Staubli VAL3: Compensated.dtx

public frame fReference = {x=1504.182, y=53.840, z=-415.791, rx=0.201, ry=-0.641, rz=0.004, fatherId=world[0]}
public jointRx jPark = {j1=0.000, j2=0.000, j3=90.000, j4=0.000, j5=90.000, j6=0.000}
public jointRx jJoint = {j1=2.01098, j2=34.80611, j3=88.39690, j4=0.21482, j5=56.14953, j6=-178.11080}
public mdesc mNomSpeed = {accel=100, vel=100, decel=100, tmax=99999, rmax=99999, blend=off, leave=50, reach=50}
public mdesc mSpeed = {tmax=33.3, rmax=100, leave=0.1, reach=0.1, blend=cartesian}
public num nTraj
num nTimeStop
num nTimeStart
num nMode
num nEtat
public pointRx pPoint[1313]
  [0] = {x=-35.000, y=0.000, z=0.000, rx=-0.000, ry=0.000, rz=-0.000, shoulder=lefty, elbow=epositive, wrist=wpositive, fatherId=fReference[0]}
  [1] = {x=-34.500, y=0.000, z=-0.007, rx=-0.000, ry=0.000, rz=-0.000, shoulder=lefty, elbow=epositive, wrist=wpositive, fatherId=fReference[0]}
  [2] = {x=-34.000, y=0.000, z=-0.014, rx=-0.000, ry=0.000, rz=-0.000, shoulder=lefty, elbow=epositive, wrist=wpositive, fatherId=fReference[0]}
  [3] = {x=-33.499, y=0.000, z=-0.022, rx=-0.000, ry=0.000, rz=-0.000, shoulder=lefty, elbow=epositive, wrist=wpositive, fatherId=fReference[0]}
  [4] = {x=-32.998, y=0.000, z=-0.029, rx=-0.000, ry=0.000, rz=-0.000, shoulder=lefty, elbow=epositive, wrist=wpositive, fatherId=fReference[0]}
  [5] = {x=-32.497, y=0.000, z=-0.036, rx=-0.000, ry=0.000, rz=-0.000, shoulder=lefty, elbow=epositive, wrist=wpositive, fatherId=fReference[0]}
  [6] = {x=-31.997, y=0.000, z=-0.044, rx=-0.000, ry=0.000, rz=-0.000, shoulder=lefty, elbow=epositive, wrist=wpositive, fatherId=fReference[0]}
  [7] = {x=-31.496, y=0.000, z=-0.051, rx=-0.000, ry=0.000, rz=-0.000, shoulder=lefty, elbow=epositive, wrist=wpositive, fatherId=fReference[0]}
  [8] = {x=-30.995, y=0.000, z=-0.059, rx=-0.000, ry=0.000, rz=-0.000, shoulder=lefty, elbow=epositive, wrist=wpositive, fatherId=fReference[0]}
  [9] = {x=-30.494, y=0.000, z=-0.066, rx=-0.000, ry=0.000, rz=-0.000, shoulder=lefty, elbow=epositive, wrist=wpositive, fatherId=fReference[0]}
  [10] = {x=-29.993, y=0.000, z=-0.073, rx=-0.000, ry=0.000, rz=-0.000, shoulder=lefty, elbow=epositive, wrist=wpositive, fatherId=fReference[0]}
  [11] = {x=-29.493, y=0.000, z=-0.081, rx=-0.000, ry=0.000, rz=-0.000, shoulder=lefty, elbow=epositive, wrist=wpositive, fatherId=fReference[0]}
  [12] = {x=-28.992, y=0.000, z=-0.088, rx=-0.000, ry=0.000, rz=-0.000, shoulder=lefty, elbow=epositive, wrist=wpositive, fatherId=fReference[0]}
  [13] = {x=-28.491, y=0.000, z=-0.095, rx=-0.000, ry=0.000, rz=-0.000, shoulder=lefty, elbow=epositive, wrist=wpositive, fatherId=fReference[0]}
  [14] = {x=-27.991, y=0.000, z=-0.103, rx=-0.000, ry=0.000, rz=-0.000, shoulder=lefty, elbow=epositive, wrist=wpositive, fatherId=fReference[0]}
  [15] = {x=-27.490, y=0.000, z=-0.110, rx=-0.000, ry=0.000, rz=-0.000, shoulder=lefty, elbow=epositive, wrist=wpositive, fatherId=fReference[0]}
  [16] = {x=-26.989, y=0.000, z=-0.117, rx=-0.000, ry=0.000, rz=-0.000, shoulder=lefty, elbow=epositive, wrist=wpositive, fatherId=fReference[0]}
  [17] = {x=-26.489, y=0.000, z=-0.125, rx=-0.000, ry=0.000, rz=-0.000, shoulder=lefty, elbow=epositive, wrist=wpositive, fatherId=fReference[0]}
  [18] = {x=-25.988, y=0.000, z=-0.132, rx=-0.000, ry=0.000, rz=-0.000, shoulder=lefty, elbow=epositive, wrist=wpositive, fatherId=fReference[0]}
  [19] = {x=-25.487, y=0.000, z=-0.139, rx=-0.000, ry=0.000, rz=-0.000, shoulder=lefty, elbow=epositive, wrist=wpositive, fatherId=fReference[0]}
  [20] = {x=-24.987, y=0.000, z=-0.147, rx=-0.000, ry=0.000, rz=-0.000, shoulder=lefty, elbow=epositive, wrist=wpositive, fatherId=fReference[0]}
  [21] = {x=-24.486, y=0.000, z=-0.154, rx=-0.000, ry=0.000, rz=-0.000, shoulder=lefty, elbow=epositive, wrist=wpositive, fatherId=fReference[0]}
  [22] = {x=-23.986, y=0.000, z=-0.161, rx=-0.000, ry=0.000, rz=-0.000, shoulder=lefty, elbow=epositive, wrist=wpositive, fatherId=fReference[0]}
  [23] = {x=-23.485, y=0.000, z=-0.169, rx=-0.000, ry=0.000, rz=-0.000, shoulder=lefty, elbow=epositive, wrist=wpositive, fatherId=fReference[0]}
  [24] = {x=-22.985, y=0.000, z=-0.176, rx=-0.000, ry=0.000, rz=-0.000, shoulder=lefty, elbow=epositive, wrist=wpositive, fatherId=fReference[0]}
  [25] = {x=-22.484, y=0.000, z=-0.183, rx=-0.000, ry=0.000, rz=-0.000, shoulder=lefty, elbow=epositive, wrist=wpositive, fatherId=fReference[0]}
  [26] = {x=-21.983, y=0.000, z=-0.191, rx=-0.000, ry=0.000, rz=-0.000, shoulder=lefty, elbow=epositive, wrist=wpositive, fatherId=fReference[0]}
  [27] = {x=-21.483, y=0.000, z=-0.198, rx=-0.000, ry=0.000, rz=-0.000, shoulder=lefty, elbow=epositive, wrist=wpositive, fatherId=fReference[0]}
  [28] = {x=-20.982, y=0.000, z=-0.205, rx=-0.000, ry=0.000, rz=-0.000, shoulder=lefty, elbow=epositive, wrist=wpositive, fatherId=fReference[0]}
  [29] = {x=-20.482, y=0.000, z=-0.213, rx=-0.000, ry=0.000, rz=-0.000, shoulder=lefty, elbow=epositive, wrist=wpositive, fatherId=fReference[0]}
  [30] = {x=-19.981, y=0.000, z=-0.220, rx=-0.000, ry=0.000, rz=-0.000, shoulder=lefty, elbow=epositive, wrist=wpositive, fatherId=fReference[0]}
  [31] = {x=-19.481, y=0.000, z=-0.227, rx=-0.000, ry=0.000, rz=-0.000, shoulder=lefty, elbow=epositive, wrist=wpositive, fatherId=fReference[0]}
  [32] = {x=-18.980, y=0.000, z=-0.234, rx=-0.000, ry=0.000, rz=-0.000, shoulder=lefty, elbow=epositive, wrist=wpositive, fatherId=fReference[0]}
  [33] = {x=-18.480, y=0.000, z=-0.242, rx=-0.000, ry=0.000, rz=-0.000, shoulder=lefty, elbow=epositive, wrist=wpositive, fatherId=fReference[0]}
  [34] = {x=-17.979, y=0.000, z=-0.249, rx=-0.000, ry=0.000, rz=-0.000, shoulder=lefty, elbow=epositive, wrist=wpositive, fatherId=fReference[0]}
  [35] = {x=-17.479, y=0.000, z=-0.256, rx=-0.000, ry=0.000, rz=-0.000, shoulder=lefty, elbow=epositive, wrist=wpositive, fatherId=fReference[0]}
  [36] = {x=-16.978, y=0.000, z=-0.264, rx=-0.000, ry=0.000, rz=-0.000, shoulder=lefty, elbow=epositive, wrist=wpositive, fatherId=fReference[0]}
  [37] = {x=-16.478, y=0.000, z=-0.271, rx=-0.000, ry=0.000, rz=-0.000, shoulder=lefty, elbow=epositive, wrist=wpositive, fatherId=fReference[0]}
  [38] = {x=-15.977, y=0.000, z=-0.278, rx=-0.000, ry=0.000, rz=-0.000, shoulder=lefty, elbow=epositive, wrist=wpositive, fatherId=fReference[0]}
  [39] = {x=-15.477, y=0.000, z=-0.285, rx=-0.000, ry=0.000, rz=-0.000, shoulder=lefty, elbow=epositive, wrist=wpositive, fatherId=fReference[0]}
  [40] = {x=-14.976, y=0.000, z=-0.293, rx=-0.000, ry=0.000, rz=-0.000, shoulder=lefty, elbow=epositive, wrist=wpositive, fatherId=fReference[0]}
  [41] = {x=-14.476, y=0.000, z=-0.300, rx=-0.000, ry=0.000, rz=-0.000, shoulder=lefty, elbow=epositive, wrist=wpositive, fatherId=fReference[0]}
  [42] = {x=-13.975, y=0.000, z=-0.307, rx=-0.000, ry=0.000, rz=-0.000, shoulder=lefty, elbow=epositive, wrist=wpositive, fatherId=fReference[0]}
  [43] = {x=-13.475, y=0.000, z=-0.315, rx=-0.000, ry=0.000, rz=-0.000, shoulder=lefty, elbow=epositive, wrist=wpositive, fatherId=fReference[0]}
  [44] = {x=-12.975, y=0.000, z=-0.322, rx=-0.000, ry=0.000, rz=-0.000, shoulder=lefty, elbow=epositive, wrist=wpositive, fatherId=fReference[0]}
  [45] = {x=-12.474, y=0.000, z=-0.329, rx=-0.000, ry=0.000, rz=-0.000, shoulder=lefty, elbow=epositive, wrist=wpositive, fatherId=fReference[0]}
  [46] = {x=-11.974, y=0.000, z=-0.336, rx=-0.000, ry=0.000, rz=-0.000, shoulder=lefty, elbow=epositive, wrist=wpositive, fatherId=fReference[0]}
  [47] = {x=-11.473, y=0.000, z=-0.344, rx=-0.000, ry=0.000, rz=-0.000, shoulder=lefty, elbow=epositive, wrist=wpositive, fatherId=fReference[0]}
  [48] = {x=-10.973, y=0.000, z=-0.351, rx=-0.000, ry=0.000, rz=-0.000, shoulder=lefty, elbow=epositive, wrist=wpositive, fatherId=fReference[0]}
  [49] = {x=-10.472, y=0.000, z=-0.358, rx=-0.000, ry=0.000, rz=-0.000, shoulder=lefty, elbow=epositive, wrist=wpositive, fatherId=fReference[0]}
  [50] = {x=-9.972, y=0.000, z=-0.366, rx=-0.000, ry=0.000, rz=-0.000, shoulder=lefty, elbow=epositive, wrist=wpositive, fatherId=fReference[0]}
  [51] = {x=-9.471, y=0.000, z=-0.373, rx=-0.000, ry=0.000, rz=-0.000, shoulder=lefty, elbow=epositive, wrist=wpositive, fatherId=fReference[0]}
  [52] = {x=-8.971, y=0.000, z=-0.380, rx=-0.000, ry=0.000, rz=-0.000, shoulder=lefty, elbow=epositive, wrist=wpositive, fatherId=fReference[0]}
  [53] = {x=-8.470, y=0.000, z=-0.388, rx=-0.000, ry=0.000, rz=-0.000, shoulder=lefty, elbow=epositive, wrist=wpositive, fatherId=fReference[0]}
  [54] = {x=-7.969, y=0.000, z=-0.395, rx=-0.000, ry=0.000, rz=-0.000, shoulder=lefty, elbow=epositive, wrist=wpositive, fatherId=fReference[0]}
  [55] = {x=-7.469, y=0.000, z=-0.402, rx=-0.000, ry=0.000, rz=-0.000, shoulder=lefty, elbow=epositive, wrist=wpositive, fatherId=fReference[0]}
  [56] = {x=-6.968, y=0.000, z=-0.409, rx=-0.000, ry=0.000, rz=-0.000, shoulder=lefty, elbow=epositive, wrist=wpositive, fatherId=fReference[0]}
  [57] = {x=-6.468, y=0.000, z=-0.417, rx=-0.000, ry=0.000, rz=-0.000, shoulder=lefty, elbow=epositive, wrist=wpositive, fatherId=fReference[0]}
  [58] = {x=-5.967, y=0.000, z=-0.424, rx=-0.000, ry=0.000, rz=-0.000, shoulder=lefty, elbow=epositive, wrist=wpositive, fatherId=fReference[0]}
  [59] = {x=-5.467, y=0.000, z=-0.431, rx=-0.000, ry=0.000, rz=-0.000, shoulder=lefty, elbow=epositive, wrist=wpositive, fatherId=fReference[0]}
  [60] = {x=-4.966, y=0.000, z=-0.439, rx=-0.000, ry=0.000, rz=-0.000, shoulder=lefty, elbow=epositive, wrist=wpositive, fatherId=fReference[0]}
  [61] = {x=-4.466, y=0.000, z=-0.446, rx=-0.000, ry=0.000, rz=-0.000, shoulder=lefty, elbow=epositive, wrist=wpositive, fatherId=fReference[0]}
  [62] = {x=-3.965, y=0.000, z=-0.453, rx=-0.000, ry=0.000, rz=-0.000, shoulder=lefty, elbow=epositive, wrist=wpositive, fatherId=fReference[0]}
  [63] = {x=-3.464, y=0.000, z=-0.461, rx=-0.000, ry=0.000, rz=-0.000, shoulder=lefty, elbow=epositive, wrist=wpositive, fatherId=fReference[0]}
  [64] = {x=-2.964, y=0.000, z=-0.468, rx=-0.000, ry=0.000, rz=-0.000, shoulder=lefty, elbow=epositive, wrist=wpositive, fatherId=fReference[0]}
  [65] = {x=-2.463, y=0.000, z=-0.475, rx=-0.000, ry=0.000, rz=-0.000, shoulder=lefty, elbow=epositive, wrist=wpositive, fatherId=fReference[0]}
  [66] = {x=-1.963, y=0.000, z=-0.483, rx=-0.000, ry=0.000, rz=-0.000, shoulder=lefty, elbow=epositive, wrist=wpositive, fatherId=fReference[0]}
  [67] = {x=-1.462, y=0.000, z=-0.490, rx=-0.000, ry=0.000, rz=-0.000, shoulder=lefty, elbow=epositive, wrist=wpositive, fatherId=fReference[0]}
  [68] = {x=-0.961, y=0.000, z=-0.497, rx=-0.000, ry=0.000, rz=-0.000, shoulder=lefty, elbow=epositive, wrist=wpositive, fatherId=fReference[0]}
  [69] = {x=-0.461, y=0.000, z=-0.505, rx=-0.000, ry=0.000, rz=-0.000, shoulder=lefty, elbow=epositive, wrist=wpositive, fatherId=fReference[0]}
  [70] = {x=0.040, y=0.000, z=-0.512, rx=-0.000, ry=0.000, rz=-0.000, shoulder=lefty, elbow=epositive, wrist=wpositive, fatherId=fReference[0]}
  [71] = {x=0.541, y=0.000, z=-0.519, rx=-0.000, ry=0.000, rz=-0.000, shoulder=lefty, elbow=epositive, wrist=wpositive, fatherId=fReference[0]}
  [72] = {x=1.041, y=0.000, z=-0.527, rx=-0.000, ry=0.000, rz=-0.000, shoulder=lefty, elbow=epositive, wrist=wpositive, fatherId=fReference[0]}
  [73] = {x=1.542, y=0.000, z=-0.534, rx=-0.000, ry=0.000, rz=-0.000, shoulder=lefty, elbow=epositive, wrist=wpositive, fatherId=fReference[0]}
  [74] = {x=2.043, y=0.000, z=-0.541, rx=-0.000, ry=0.000, rz=-0.000, shoulder=lefty, elbow=epositive, wrist=wpositive, fatherId=fReference[0]}
  [75] = {x=2.544, y=0.000, z=-0.549, rx=-0.000, ry=0.000, rz=-0.000, shoulder=lefty, elbow=epositive, wrist=wpositive, fatherId=fReference[0]}
  [76] = {x=3.044, y=0.000, z=-0.556, rx=-0.000, ry=0.000, rz=-0.000, shoulder=lefty, elbow=epositive, wrist=wpositive, fatherId=fReference[0]}
  [77] = {x=3.545, y=0.000, z=-0.563, rx=-0.000, ry=0.000, rz=-0.000, shoulder=lefty, elbow=epositive, wrist=wpositive, fatherId=fReference[0]}
  [78] = {x=4.046, y=0.000, z=-0.571, rx=-0.000, ry=0.000, rz=-0.000, shoulder=lefty, elbow=epositive, wrist=wpositive, fatherId=fReference[0]}
  [79] = {x=4.547, y=0.000, z=-0.578, rx=-0.000, ry=0.000, rz=-0.000, shoulder=lefty, elbow=epositive, wrist=wpositive, fatherId=fReference[0]}
  [80] = {x=5.047, y=0.000, z=-0.586, rx=-0.000, ry=0.000, rz=-0.000, shoulder=lefty, elbow=epositive, wrist=wpositive, fatherId=fReference[0]}
  [81] = {x=5.548, y=0.000, z=-0.593, rx=-0.000, ry=0.000, rz=-0.000, shoulder=lefty, elbow=epositive, wrist=wpositive, fatherId=fReference[0]}
  [82] = {x=6.049, y=0.000, z=-0.600, rx=-0.000, ry=0.000, rz=-0.000, shoulder=lefty, elbow=epositive, wrist=wpositive, fatherId=fReference[0]}
  [83] = {x=6.550, y=0.000, z=-0.608, rx=-0.000, ry=0.000, rz=-0.000, shoulder=lefty, elbow=epositive, wrist=wpositive, fatherId=fReference[0]}
  [84] = {x=7.051, y=0.000, z=-0.615, rx=-0.000, ry=0.000, rz=-0.000, shoulder=lefty, elbow=epositive, wrist=wpositive, fatherId=fReference[0]}
  [85] = {x=7.552, y=0.000, z=-0.623, rx=-0.000, ry=0.000, rz=-0.000, shoulder=lefty, elbow=epositive, wrist=wpositive, fatherId=fReference[0]}
  [86] = {x=8.053, y=0.000, z=-0.630, rx=-0.000, ry=0.000, rz=-0.000, shoulder=lefty, elbow=epositive, wrist=wpositive, fatherId=fReference[0]}
  [87] = {x=8.554, y=0.000, z=-0.637, rx=-0.000, ry=0.000, rz=-0.000, shoulder=lefty, elbow=epositive, wrist=wpositive, fatherId=fReference[0]}
  [88] = {x=9.055, y=0.000, z=-0.645, rx=-0.000, ry=0.000, rz=-0.000, shoulder=lefty, elbow=epositive, wrist=wpositive, fatherId=fReference[0]}
  [89] = {x=9.556, y=0.000, z=-0.652, rx=-0.000, ry=0.000, rz=-0.000, shoulder=lefty, elbow=epositive, wrist=wpositive, fatherId=fReference[0]}
  [90] = {x=10.057, y=0.000, z=-0.660, rx=-0.000, ry=0.000, rz=-0.000, shoulder=lefty, elbow=epositive, wrist=wpositive, fatherId=fReference[0]}
  [91] = {x=10.558, y=0.000, z=-0.667, rx=-0.000, ry=0.000, rz=-0.000, shoulder=lefty, elbow=epositive, wrist=wpositive, fatherId=fReference[0]}
  [92] = {x=11.059, y=0.000, z=-0.675, rx=-0.000, ry=0.000, rz=-0.000, shoulder=lefty, elbow=epositive, wrist=wpositive, fatherId=fReference[0]}
  [93] = {x=11.560, y=0.000, z=-0.682, rx=-0.000, ry=0.000, rz=-0.000, shoulder=lefty, elbow=epositive, wrist=wpositive, fatherId=fReference[0]}
  [94] = {x=12.061, y=0.000, z=-0.690, rx=-0.000, ry=0.000, rz=-0.000, shoulder=lefty, elbow=epositive, wrist=wpositive, fatherId=fReference[0]}
  [95] = {x=12.562, y=0.000, z=-0.697, rx=-0.000, ry=0.000, rz=-0.000, shoulder=lefty, elbow=epositive, wrist=wpositive, fatherId=fReference[0]}
  [96] = {x=13.064, y=0.000, z=-0.705, rx=-0.000, ry=0.000, rz=-0.000, shoulder=lefty, elbow=epositive, wrist=wpositive, fatherId=fReference[0]}
  [97] = {x=13.565, y=0.000, z=-0.712, rx=-0.000, ry=0.000, rz=-0.000, shoulder=lefty, elbow=epositive, wrist=wpositive, fatherId=fReference[0]}
  [98] = {x=14.066, y=0.000, z=-0.720, rx=-0.000, ry=0.000, rz=-0.000, shoulder=lefty, elbow=epositive, wrist=wpositive, fatherId=fReference[0]}
  [99] = {x=14.567, y=0.000, z=-0.727, rx=-0.000, ry=0.000, rz=-0.000, shoulder=lefty, elbow=epositive, wrist=wpositive, fatherId=fReference[0]}
  [100] = {x=15.069, y=0.000, z=-0.735, rx=-0.000, ry=0.000, rz=-0.000, shoulder=lefty, elbow=epositive, wrist=wpositive, fatherId=fReference[0]}
  [101] = {x=15.570, y=0.000, z=-0.742, rx=-0.000, ry=0.000, rz=-0.000, shoulder=lefty, elbow=epositive, wrist=wpositive, fatherId=fReference[0]}
  [102] = {x=16.071, y=0.000, z=-0.750, rx=-0.000, ry=0.000, rz=-0.000, shoulder=lefty, elbow=epositive, wrist=wpositive, fatherId=fReference[0]}
  [103] = {x=16.573, y=0.000, z=-0.757, rx=-0.000, ry=0.000, rz=-0.000, shoulder=lefty, elbow=epositive, wrist=wpositive, fatherId=fReference[0]}
  [104] = {x=17.074, y=0.000, z=-0.765, rx=-0.000, ry=0.000, rz=-0.000, shoulder=lefty, elbow=epositive, wrist=wpositive, fatherId=fReference[0]}
  [105] = {x=17.576, y=0.000, z=-0.772, rx=-0.000, ry=0.000, rz=-0.000, shoulder=lefty, elbow=epositive, wrist=wpositive, fatherId=fReference[0]}
  [106] = {x=18.077, y=0.000, z=-0.780, rx=-0.000, ry=0.000, rz=-0.000, shoulder=lefty, elbow=epositive, wrist=wpositive, fatherId=fReference[0]}
  [107] = {x=18.579, y=0.000, z=-0.788, rx=-0.000, ry=0.000, rz=-0.000, shoulder=lefty, elbow=epositive, wrist=wpositive, fatherId=fReference[0]}
  [108] = {x=19.081, y=0.000, z=-0.795, rx=-0.000, ry=0.000, rz=-0.000, shoulder=lefty, elbow=epositive, wrist=wpositive, fatherId=fReference[0]}
  [109] = {x=19.582, y=0.000, z=-0.803, rx=-0.000, ry=0.000, rz=-0.000, shoulder=lefty, elbow=epositive, wrist=wpositive, fatherId=fReference[0]}
  [110] = {x=20.084, y=0.000, z=-0.811, rx=-0.000, ry=0.000, rz=-0.000, shoulder=lefty, elbow=epositive, wrist=wpositive, fatherId=fReference[0]}
  [111] = {x=20.586, y=0.000, z=-0.818, rx=-0.000, ry=0.000, rz=-0.000, shoulder=lefty, elbow=epositive, wrist=wpositive, fatherId=fReference[0]}
  [112] = {x=21.088, y=0.000, z=-0.826, rx=-0.000, ry=0.000, rz=-0.000, shoulder=lefty, elbow=epositive, wrist=wpositive, fatherId=fReference[0]}
  [113] = {x=21.589, y=0.000, z=-0.834, rx=-0.000, ry=0.000, rz=-0.000, shoulder=lefty, elbow=epositive, wrist=wpositive, fatherId=fReference[0]}
  [114] = {x=22.091, y=0.000, z=-0.841, rx=-0.000, ry=0.000, rz=-0.000, shoulder=lefty, elbow=epositive, wrist=wpositive, fatherId=fReference[0]}
  [115] = {x=22.593, y=0.000, z=-0.849, rx=-0.000, ry=0.000, rz=-0.000, shoulder=lefty, elbow=epositive, wrist=wpositive, fatherId=fReference[0]}
  [116] = {x=23.095, y=0.000, z=-0.857, rx=-0.000, ry=0.000, rz=-0.000, shoulder=lefty, elbow=epositive, wrist=wpositive, fatherId=fReference[0]}
  [117] = {x=23.597, y=0.000, z=-0.864, rx=-0.000, ry=0.000, rz=-0.000, shoulder=lefty, elbow=epositive, wrist=wpositive, fatherId=fReference[0]}
  [118] = {x=24.100, y=0.000, z=-0.872, rx=-0.000, ry=0.000, rz=-0.000, shoulder=lefty, elbow=epositive, wrist=wpositive, fatherId=fReference[0]}
  [119] = {x=24.602, y=0.000, z=-0.880, rx=-0.000, ry=0.000, rz=-0.000, shoulder=lefty, elbow=epositive, wrist=wpositive, fatherId=fReference[0]}
  [120] = {x=25.104, y=0.000, z=-0.888, rx=-0.000, ry=0.000, rz=-0.000, shoulder=lefty, elbow=epositive, wrist=wpositive, fatherId=fReference[0]}
  [121] = {x=25.606, y=0.000, z=-0.896, rx=-0.000, ry=0.000, rz=-0.000, shoulder=lefty, elbow=epositive, wrist=wpositive, fatherId=fReference[0]}
  [122] = {x=26.108, y=0.000, z=-0.903, rx=-0.000, ry=0.000, rz=-0.000, shoulder=lefty, elbow=epositive, wrist=wpositive, fatherId=fReference[0]}
  [123] = {x=26.611, y=0.000, z=-0.911, rx=-0.000, ry=0.000, rz=-0.000, shoulder=lefty, elbow=epositive, wrist=wpositive, fatherId=fReference[0]}
  [124] = {x=27.113, y=0.000, z=-0.919, rx=-0.000, ry=0.000, rz=-0.000, shoulder=lefty, elbow=epositive, wrist=wpositive, fatherId=fReference[0]}
  [125] = {x=27.616, y=0.000, z=-0.927, rx=-0.000, ry=0.000, rz=-0.000, shoulder=lefty, elbow=epositive, wrist=wpositive, fatherId=fReference[0]}
  [126] = {x=28.118, y=0.000, z=-0.935, rx=-0.000, ry=0.000, rz=-0.000, shoulder=lefty, elbow=epositive, wrist=wpositive, fatherId=fReference[0]}
  [127] = {x=28.621, y=0.000, z=-0.943, rx=-0.000, ry=0.000, rz=-0.000, shoulder=lefty, elbow=epositive, wrist=wpositive, fatherId=fReference[0]}
  [128] = {x=29.124, y=0.000, z=-0.951, rx=-0.000, ry=0.000, rz=-0.000, shoulder=lefty, elbow=epositive, wrist=wpositive, fatherId=fReference[0]}
  [129] = {x=29.627, y=0.000, z=-0.959, rx=-0.000, ry=0.000, rz=-0.000, shoulder=lefty, elbow=epositive, wrist=wpositive, fatherId=fReference[0]}
  [130] = {x=30.130, y=0.000, z=-0.967, rx=-0.000, ry=0.000, rz=-0.000, shoulder=lefty, elbow=epositive, wrist=wpositive, fatherId=fReference[0]}
  [131] = {x=30.633, y=0.000, z=-0.975, rx=-0.000, ry=0.000, rz=-0.000, shoulder=lefty, elbow=epositive, wrist=wpositive, fatherId=fReference[0]}
  [132] = {x=31.136, y=0.000, z=-0.983, rx=-0.000, ry=0.000, rz=-0.000, shoulder=lefty, elbow=epositive, wrist=wpositive, fatherId=fReference[0]}
  [133] = {x=31.639, y=0.000, z=-0.991, rx=-0.000, ry=0.000, rz=-0.000, shoulder=lefty, elbow=epositive, wrist=wpositive, fatherId=fReference[0]}
  [134] = {x=32.142, y=0.000, z=-0.999, rx=-0.000, ry=0.000, rz=-0.000, shoulder=lefty, elbow=epositive, wrist=wpositive, fatherId=fReference[0]}
  [135] = {x=32.646, y=0.000, z=-1.007, rx=-0.000, ry=0.000, rz=-0.000, shoulder=lefty, elbow=epositive, wrist=wpositive, fatherId=fReference[0]}
  [136] = {x=33.149, y=0.000, z=-1.015, rx=-0.000, ry=0.000, rz=-0.000, shoulder=lefty, elbow=epositive, wrist=wpositive, fatherId=fReference[0]}
  [137] = {x=33.653, y=0.000, z=-1.023, rx=-0.000, ry=0.000, rz=-0.000, shoulder=lefty, elbow=epositive, wrist=wpositive, fatherId=fReference[0]}
  [138] = {x=34.156, y=0.000, z=-1.031, rx=-0.000, ry=0.000, rz=-0.000, shoulder=lefty, elbow=epositive, wrist=wpositive, fatherId=fReference[0]}
  [139] = {x=34.660, y=0.000, z=-1.040, rx=-0.000, ry=0.000, rz=-0.000, shoulder=lefty, elbow=epositive, wrist=wpositive, fatherId=fReference[0]}
  [140] = {x=35.164, y=0.000, z=-1.048, rx=-0.000, ry=0.000, rz=-0.000, shoulder=lefty, elbow=epositive, wrist=wpositive, fatherId=fReference[0]}
  [141] = {x=34.634, y=0.000, z=-1.057, rx=-0.000, ry=0.000, rz=-0.000, shoulder=lefty, elbow=epositive, wrist=wpositive, fatherId=fReference[0]}
  [142] = {x=34.132, y=0.000, z=-1.063, rx=-0.000, ry=0.000, rz=-0.000, shoulder=lefty, elbow=epositive, wrist=wpositive, fatherId=fReference[0]}
  [143] = {x=33.631, y=0.000, z=-1.070, rx=-0.000, ry=0.000, rz=-0.000, shoulder=lefty, elbow=epositive, wrist=wpositive, fatherId=fReference[0]}
  [144] = {x=33.130, y=0.000, z=-1.077, rx=-0.000, ry=0.000, rz=-0.000, shoulder=lefty, elbow=epositive, wrist=wpositive, fatherId=fReference[0]}
  [145] = {x=32.628, y=0.000, z=-1.084, rx=-0.000, ry=0.000, rz=-0.000, shoulder=lefty, elbow=epositive, wrist=wpositive, fatherId=fReference[0]}
  [146] = {x=32.127, y=0.000, z=-1.091, rx=-0.000, ry=0.000, rz=-0.000, shoulder=lefty, elbow=epositive, wrist=wpositive, fatherId=fReference[0]}
  [147] = {x=31.626, y=0.000, z=-1.098, rx=-0.000, ry=0.000, rz=-0.000, shoulder=lefty, elbow=epositive, wrist=wpositive, fatherId=fReference[0]}
  [148] = {x=31.126, y=0.000, z=-1.105, rx=-0.000, ry=0.000, rz=-0.000, shoulder=lefty, elbow=epositive, wrist=wpositive, fatherId=fReference[0]}
  [149] = {x=30.625, y=0.000, z=-1.112, rx=-0.000, ry=0.000, rz=-0.000, shoulder=lefty, elbow=epositive, wrist=wpositive, fatherId=fReference[0]}
  [150] = {x=30.124, y=0.000, z=-1.119, rx=-0.000, ry=0.000, rz=-0.000, shoulder=lefty, elbow=epositive, wrist=wpositive, fatherId=fReference[0]}
  [151] = {x=29.624, y=0.000, z=-1.126, rx=-0.000, ry=0.000, rz=-0.000, shoulder=lefty, elbow=epositive, wrist=wpositive, fatherId=fReference[0]}
  [152] = {x=29.123, y=0.000, z=-1.133, rx=-0.000, ry=0.000, rz=-0.000, shoulder=lefty, elbow=epositive, wrist=wpositive, fatherId=fReference[0]}
  [153] = {x=28.622, y=0.000, z=-1.140, rx=-0.000, ry=0.000, rz=-0.000, shoulder=lefty, elbow=epositive, wrist=wpositive, fatherId=fReference[0]}
  [154] = {x=28.122, y=0.000, z=-1.147, rx=-0.000, ry=0.000, rz=-0.000, shoulder=lefty, elbow=epositive, wrist=wpositive, fatherId=fReference[0]}
  [155] = {x=27.621, y=0.000, z=-1.154, rx=-0.000, ry=0.000, rz=-0.000, shoulder=lefty, elbow=epositive, wrist=wpositive, fatherId=fReference[0]}
  [156] = {x=27.121, y=0.000, z=-1.161, rx=-0.000, ry=0.000, rz=-0.000, shoulder=lefty, elbow=epositive, wrist=wpositive, fatherId=fReference[0]}
  [157] = {x=26.621, y=0.000, z=-1.169, rx=-0.000, ry=0.000, rz=-0.000, shoulder=lefty, elbow=epositive, wrist=wpositive, fatherId=fReference[0]}
  [158] = {x=26.120, y=0.000, z=-1.176, rx=-0.000, ry=0.000, rz=-0.000, shoulder=lefty, elbow=epositive, wrist=wpositive, fatherId=fReference[0]}
  [159] = {x=25.620, y=0.000, z=-1.183, rx=-0.000, ry=0.000, rz=-0.000, shoulder=lefty, elbow=epositive, wrist=wpositive, fatherId=fReference[0]}
  [160] = {x=25.120, y=0.000, z=-1.190, rx=-0.000, ry=0.000, rz=-0.000, shoulder=lefty, elbow=epositive, wrist=wpositive, fatherId=fReference[0]}
  [161] = {x=24.619, y=0.000, z=-1.197, rx=-0.000, ry=0.000, rz=-0.000, shoulder=lefty, elbow=epositive, wrist=wpositive, fatherId=fReference[0]}
  [162] = {x=24.119, y=0.000, z=-1.204, rx=-0.000, ry=0.000, rz=-0.000, shoulder=lefty, elbow=epositive, wrist=wpositive, fatherId=fReference[0]}
  [163] = {x=23.619, y=0.000, z=-1.212, rx=-0.000, ry=0.000, rz=-0.000, shoulder=lefty, elbow=epositive, wrist=wpositive, fatherId=fReference[0]}
  [164] = {x=23.119, y=0.000, z=-1.219, rx=-0.000, ry=0.000, rz=-0.000, shoulder=lefty, elbow=epositive, wrist=wpositive, fatherId=fReference[0]}
  [165] = {x=22.618, y=0.000, z=-1.226, rx=-0.000, ry=0.000, rz=-0.000, shoulder=lefty, elbow=epositive, wrist=wpositive, fatherId=fReference[0]}
  [166] = {x=22.118, y=0.000, z=-1.233, rx=-0.000, ry=0.000, rz=-0.000, shoulder=lefty, elbow=epositive, wrist=wpositive, fatherId=fReference[0]}
  [167] = {x=21.618, y=0.000, z=-1.240, rx=-0.000, ry=0.000, rz=-0.000, shoulder=lefty, elbow=epositive, wrist=wpositive, fatherId=fReference[0]}
  [168] = {x=21.118, y=0.000, z=-1.248, rx=-0.000, ry=0.000, rz=-0.000, shoulder=lefty, elbow=epositive, wrist=wpositive, fatherId=fReference[0]}
  [169] = {x=20.618, y=0.000, z=-1.255, rx=-0.000, ry=0.000, rz=-0.000, shoulder=lefty, elbow=epositive, wrist=wpositive, fatherId=fReference[0]}
  [170] = {x=20.118, y=0.000, z=-1.262, rx=-0.000, ry=0.000, rz=-0.000, shoulder=lefty, elbow=epositive, wrist=wpositive, fatherId=fReference[0]}
  [171] = {x=19.618, y=0.000, z=-1.269, rx=-0.000, ry=0.000, rz=-0.000, shoulder=lefty, elbow=epositive, wrist=wpositive, fatherId=fReference[0]}
  [172] = {x=19.118, y=0.000, z=-1.276, rx=-0.000, ry=0.000, rz=-0.000, shoulder=lefty, elbow=epositive, wrist=wpositive, fatherId=fReference[0]}
  [173] = {x=18.618, y=0.000, z=-1.284, rx=-0.000, ry=0.000, rz=-0.000, shoulder=lefty, elbow=epositive, wrist=wpositive, fatherId=fReference[0]}
  [174] = {x=18.118, y=0.000, z=-1.291, rx=-0.000, ry=0.000, rz=-0.000, shoulder=lefty, elbow=epositive, wrist=wpositive, fatherId=fReference[0]}
  [175] = {x=17.618, y=0.000, z=-1.298, rx=-0.000, ry=0.000, rz=-0.000, shoulder=lefty, elbow=epositive, wrist=wpositive, fatherId=fReference[0]}
  [176] = {x=17.118, y=0.000, z=-1.306, rx=-0.000, ry=0.000, rz=-0.000, shoulder=lefty, elbow=epositive, wrist=wpositive, fatherId=fReference[0]}
  [177] = {x=16.618, y=0.000, z=-1.313, rx=-0.000, ry=0.000, rz=-0.000, shoulder=lefty, elbow=epositive, wrist=wpositive, fatherId=fReference[0]}
  [178] = {x=16.118, y=0.000, z=-1.320, rx=-0.000, ry=0.000, rz=-0.000, shoulder=lefty, elbow=epositive, wrist=wpositive, fatherId=fReference[0]}
  [179] = {x=15.618, y=0.000, z=-1.327, rx=-0.000, ry=0.000, rz=-0.000, shoulder=lefty, elbow=epositive, wrist=wpositive, fatherId=fReference[0]}
  [180] = {x=15.119, y=0.000, z=-1.335, rx=-0.000, ry=0.000, rz=-0.000, shoulder=lefty, elbow=epositive, wrist=wpositive, fatherId=fReference[0]}
  [181] = {x=14.619, y=0.000, z=-1.342, rx=-0.000, ry=0.000, rz=-0.000, shoulder=lefty, elbow=epositive, wrist=wpositive, fatherId=fReference[0]}
  [182] = {x=14.119, y=0.000, z=-1.349, rx=-0.000, ry=0.000, rz=-0.000, shoulder=lefty, elbow=epositive, wrist=wpositive, fatherId=fReference[0]}
  [183] = {x=13.619, y=0.000, z=-1.357, rx=-0.000, ry=0.000, rz=-0.000, shoulder=lefty, elbow=epositive, wrist=wpositive, fatherId=fReference[0]}
  [184] = {x=13.120, y=0.000, z=-1.364, rx=-0.000, ry=0.000, rz=-0.000, shoulder=lefty, elbow=epositive, wrist=wpositive, fatherId=fReference[0]}
  [185] = {x=12.620, y=0.000, z=-1.372, rx=-0.000, ry=0.000, rz=-0.000, shoulder=lefty, elbow=epositive, wrist=wpositive, fatherId=fReference[0]}
  [186] = {x=12.120, y=0.000, z=-1.379, rx=-0.000, ry=0.000, rz=-0.000, shoulder=lefty, elbow=epositive, wrist=wpositive, fatherId=fReference[0]}
  [187] = {x=11.620, y=0.000, z=-1.386, rx=-0.000, ry=0.000, rz=-0.000, shoulder=lefty, elbow=epositive, wrist=wpositive, fatherId=fReference[0]}
  [188] = {x=11.121, y=0.000, z=-1.394, rx=-0.000, ry=0.000, rz=-0.000, shoulder=lefty, elbow=epositive, wrist=wpositive, fatherId=fReference[0]}
  [189] = {x=10.621, y=0.000, z=-1.401, rx=-0.000, ry=0.000, rz=-0.000, shoulder=lefty, elbow=epositive, wrist=wpositive, fatherId=fReference[0]}
  [190] = {x=10.121, y=0.000, z=-1.409, rx=-0.000, ry=0.000, rz=-0.000, shoulder=lefty, elbow=epositive, wrist=wpositive, fatherId=fReference[0]}
  [191] = {x=9.622, y=0.000, z=-1.416, rx=-0.000, ry=0.000, rz=-0.000, shoulder=lefty, elbow=epositive, wrist=wpositive, fatherId=fReference[0]}
  [192] = {x=9.122, y=0.000, z=-1.423, rx=-0.000, ry=0.000, rz=-0.000, shoulder=lefty, elbow=epositive, wrist=wpositive, fatherId=fReference[0]}
  [193] = {x=8.623, y=0.000, z=-1.431, rx=-0.000, ry=0.000, rz=-0.000, shoulder=lefty, elbow=epositive, wrist=wpositive, fatherId=fReference[0]}
  [194] = {x=8.123, y=0.000, z=-1.438, rx=-0.000, ry=0.000, rz=-0.000, shoulder=lefty, elbow=epositive, wrist=wpositive, fatherId=fReference[0]}
  [195] = {x=7.624, y=0.000, z=-1.446, rx=-0.000, ry=0.000, rz=-0.000, shoulder=lefty, elbow=epositive, wrist=wpositive, fatherId=fReference[0]}
  [196] = {x=7.124, y=0.000, z=-1.453, rx=-0.000, ry=0.000, rz=-0.000, shoulder=lefty, elbow=epositive, wrist=wpositive, fatherId=fReference[0]}
  [197] = {x=6.625, y=0.000, z=-1.461, rx=-0.000, ry=0.000, rz=-0.000, shoulder=lefty, elbow=epositive, wrist=wpositive, fatherId=fReference[0]}
  [198] = {x=6.125, y=0.000, z=-1.468, rx=-0.000, ry=0.000, rz=-0.000, shoulder=lefty, elbow=epositive, wrist=wpositive, fatherId=fReference[0]}
  [199] = {x=5.626, y=0.000, z=-1.476, rx=-0.000, ry=0.000, rz=-0.000, shoulder=lefty, elbow=epositive, wrist=wpositive, fatherId=fReference[0]}
  [200] = {x=5.126, y=0.000, z=-1.483, rx=-0.000, ry=0.000, rz=-0.000, shoulder=lefty, elbow=epositive, wrist=wpositive, fatherId=fReference[0]}
  [201] = {x=4.627, y=0.000, z=-1.490, rx=-0.000, ry=0.000, rz=-0.000, shoulder=lefty, elbow=epositive, wrist=wpositive, fatherId=fReference[0]}
  [202] = {x=4.127, y=0.000, z=-1.498, rx=-0.000, ry=0.000, rz=-0.000, shoulder=lefty, elbow=epositive, wrist=wpositive, fatherId=fReference[0]}
  [203] = {x=3.628, y=0.000, z=-1.506, rx=-0.000, ry=0.000, rz=-0.000, shoulder=lefty, elbow=epositive, wrist=wpositive, fatherId=fReference[0]}
  [204] = {x=3.129, y=0.000, z=-1.513, rx=-0.000, ry=0.000, rz=-0.000, shoulder=lefty, elbow=epositive, wrist=wpositive, fatherId=fReference[0]}
  [205] = {x=2.629, y=0.000, z=-1.521, rx=-0.000, ry=0.000, rz=-0.000, shoulder=lefty, elbow=epositive, wrist=wpositive, fatherId=fReference[0]}
  [206] = {x=2.130, y=0.000, z=-1.528, rx=-0.000, ry=0.000, rz=-0.000, shoulder=lefty, elbow=epositive, wrist=wpositive, fatherId=fReference[0]}
  [207] = {x=1.631, y=0.000, z=-1.536, rx=-0.000, ry=0.000, rz=-0.000, shoulder=lefty, elbow=epositive, wrist=wpositive, fatherId=fReference[0]}
  [208] = {x=1.131, y=0.000, z=-1.543, rx=-0.000, ry=0.000, rz=-0.000, shoulder=lefty, elbow=epositive, wrist=wpositive, fatherId=fReference[0]}
  [209] = {x=0.632, y=0.000, z=-1.551, rx=-0.000, ry=0.000, rz=-0.000, shoulder=lefty, elbow=epositive, wrist=wpositive, fatherId=fReference[0]}
  [210] = {x=0.133, y=0.000, z=-1.558, rx=-0.000, ry=0.000, rz=-0.000, shoulder=lefty, elbow=epositive, wrist=wpositive, fatherId=fReference[0]}
  [211] = {x=-0.366, y=0.000, z=-1.566, rx=-0.000, ry=0.000, rz=-0.000, shoulder=lefty, elbow=epositive, wrist=wpositive, fatherId=fReference[0]}
  [212] = {x=-0.865, y=0.000, z=-1.574, rx=-0.000, ry=0.000, rz=-0.000, shoulder=lefty, elbow=epositive, wrist=wpositive, fatherId=fReference[0]}
  [213] = {x=-1.364, y=0.000, z=-1.581, rx=-0.000, ry=0.000, rz=-0.000, shoulder=lefty, elbow=epositive, wrist=wpositive, fatherId=fReference[0]}
  [214] = {x=-1.864, y=0.000, z=-1.589, rx=-0.000, ry=0.000, rz=-0.000, shoulder=lefty, elbow=epositive, wrist=wpositive, fatherId=fReference[0]}
  [215] = {x=-2.363, y=0.000, z=-1.597, rx=-0.000, ry=0.000, rz=-0.000, shoulder=lefty, elbow=epositive, wrist=wpositive, fatherId=fReference[0]}
  [216] = {x=-2.862, y=0.000, z=-1.604, rx=-0.000, ry=0.000, rz=-0.000, shoulder=lefty, elbow=epositive, wrist=wpositive, fatherId=fReference[0]}
  [217] = {x=-3.361, y=0.000, z=-1.612, rx=-0.000, ry=0.000, rz=-0.000, shoulder=lefty, elbow=epositive, wrist=wpositive, fatherId=fReference[0]}
  [218] = {x=-3.859, y=0.000, z=-1.620, rx=-0.000, ry=0.000, rz=-0.000, shoulder=lefty, elbow=epositive, wrist=wpositive, fatherId=fReference[0]}
  [219] = {x=-4.358, y=0.000, z=-1.627, rx=-0.000, ry=0.000, rz=-0.000, shoulder=lefty, elbow=epositive, wrist=wpositive, fatherId=fReference[0]}
  [220] = {x=-4.857, y=0.000, z=-1.635, rx=-0.000, ry=0.000, rz=-0.000, shoulder=lefty, elbow=epositive, wrist=wpositive, fatherId=fReference[0]}
  [221] = {x=-5.356, y=0.000, z=-1.643, rx=-0.000, ry=0.000, rz=-0.000, shoulder=lefty, elbow=epositive, wrist=wpositive, fatherId=fReference[0]}
  [222] = {x=-5.855, y=0.000, z=-1.650, rx=-0.000, ry=0.000, rz=-0.000, shoulder=lefty, elbow=epositive, wrist=wpositive, fatherId=fReference[0]}
  [223] = {x=-6.354, y=0.000, z=-1.658, rx=-0.000, ry=0.000, rz=-0.000, shoulder=lefty, elbow=epositive, wrist=wpositive, fatherId=fReference[0]}
  [224] = {x=-6.853, y=0.000, z=-1.666, rx=-0.000, ry=0.000, rz=-0.000, shoulder=lefty, elbow=epositive, wrist=wpositive, fatherId=fReference[0]}
  [225] = {x=-7.351, y=0.000, z=-1.674, rx=-0.000, ry=0.000, rz=-0.000, shoulder=lefty, elbow=epositive, wrist=wpositive, fatherId=fReference[0]}
  [226] = {x=-7.850, y=0.000, z=-1.681, rx=-0.000, ry=0.000, rz=-0.000, shoulder=lefty, elbow=epositive, wrist=wpositive, fatherId=fReference[0]}
  [227] = {x=-8.349, y=0.000, z=-1.689, rx=-0.000, ry=0.000, rz=-0.000, shoulder=lefty, elbow=epositive, wrist=wpositive, fatherId=fReference[0]}
  [228] = {x=-8.848, y=0.000, z=-1.697, rx=-0.000, ry=0.000, rz=-0.000, shoulder=lefty, elbow=epositive, wrist=wpositive, fatherId=fReference[0]}
  [229] = {x=-9.346, y=0.000, z=-1.705, rx=-0.000, ry=0.000, rz=-0.000, shoulder=lefty, elbow=epositive, wrist=wpositive, fatherId=fReference[0]}
  [230] = {x=-9.845, y=0.000, z=-1.713, rx=-0.000, ry=0.000, rz=-0.000, shoulder=lefty, elbow=epositive, wrist=wpositive, fatherId=fReference[0]}
  [231] = {x=-10.343, y=0.000, z=-1.721, rx=-0.000, ry=0.000, rz=-0.000, shoulder=lefty, elbow=epositive, wrist=wpositive, fatherId=fReference[0]}
  [232] = {x=-10.842, y=0.000, z=-1.728, rx=-0.000, ry=0.000, rz=-0.000, shoulder=lefty, elbow=epositive, wrist=wpositive, fatherId=fReference[0]}
  [233] = {x=-11.341, y=0.000, z=-1.736, rx=-0.000, ry=0.000, rz=-0.000, shoulder=lefty, elbow=epositive, wrist=wpositive, fatherId=fReference[0]}
  [234] = {x=-11.839, y=0.000, z=-1.744, rx=-0.000, ry=0.000, rz=-0.000, shoulder=lefty, elbow=epositive, wrist=wpositive, fatherId=fReference[0]}
  [235] = {x=-12.338, y=0.000, z=-1.752, rx=-0.000, ry=0.000, rz=-0.000, shoulder=lefty, elbow=epositive, wrist=wpositive, fatherId=fReference[0]}
  [236] = {x=-12.836, y=0.000, z=-1.760, rx=-0.000, ry=0.000, rz=-0.000, shoulder=lefty, elbow=epositive, wrist=wpositive, fatherId=fReference[0]}
  [237] = {x=-13.334, y=0.000, z=-1.768, rx=-0.000, ry=0.000, rz=-0.000, shoulder=lefty, elbow=epositive, wrist=wpositive, fatherId=fReference[0]}
  [238] = {x=-13.833, y=0.000, z=-1.776, rx=-0.000, ry=0.000, rz=-0.000, shoulder=lefty, elbow=epositive, wrist=wpositive, fatherId=fReference[0]}
  [239] = {x=-14.331, y=0.000, z=-1.784, rx=-0.000, ry=0.000, rz=-0.000, shoulder=lefty, elbow=epositive, wrist=wpositive, fatherId=fReference[0]}
  [240] = {x=-14.829, y=0.000, z=-1.792, rx=-0.000, ry=0.000, rz=-0.000, shoulder=lefty, elbow=epositive, wrist=wpositive, fatherId=fReference[0]}
  [241] = {x=-15.328, y=0.000, z=-1.800, rx=-0.000, ry=0.000, rz=-0.000, shoulder=lefty, elbow=epositive, wrist=wpositive, fatherId=fReference[0]}
  [242] = {x=-15.826, y=0.000, z=-1.808, rx=-0.000, ry=0.000, rz=-0.000, shoulder=lefty, elbow=epositive, wrist=wpositive, fatherId=fReference[0]}
  [243] = {x=-16.324, y=0.000, z=-1.816, rx=-0.000, ry=0.000, rz=-0.000, shoulder=lefty, elbow=epositive, wrist=wpositive, fatherId=fReference[0]}
  [244] = {x=-16.822, y=0.000, z=-1.824, rx=-0.000, ry=0.000, rz=-0.000, shoulder=lefty, elbow=epositive, wrist=wpositive, fatherId=fReference[0]}
  [245] = {x=-17.320, y=0.000, z=-1.832, rx=-0.000, ry=0.000, rz=-0.000, shoulder=lefty, elbow=epositive, wrist=wpositive, fatherId=fReference[0]}
  [246] = {x=-17.818, y=0.000, z=-1.841, rx=-0.000, ry=0.000, rz=-0.000, shoulder=lefty, elbow=epositive, wrist=wpositive, fatherId=fReference[0]}
  [247] = {x=-18.316, y=0.000, z=-1.849, rx=-0.000, ry=0.000, rz=-0.000, shoulder=lefty, elbow=epositive, wrist=wpositive, fatherId=fReference[0]}
  [248] = {x=-18.814, y=0.000, z=-1.857, rx=-0.000, ry=0.000, rz=-0.000, shoulder=lefty, elbow=epositive, wrist=wpositive, fatherId=fReference[0]}
  [249] = {x=-19.311, y=0.000, z=-1.865, rx=-0.000, ry=0.000, rz=-0.000, shoulder=lefty, elbow=epositive, wrist=wpositive, fatherId=fReference[0]}
  [250] = {x=-19.809, y=0.000, z=-1.873, rx=-0.000, ry=0.000, rz=-0.000, shoulder=lefty, elbow=epositive, wrist=wpositive, fatherId=fReference[0]}
  [251] = {x=-20.307, y=0.000, z=-1.882, rx=-0.000, ry=0.000, rz=-0.000, shoulder=lefty, elbow=epositive, wrist=wpositive, fatherId=fReference[0]}
  [252] = {x=-20.804, y=0.000, z=-1.890, rx=-0.000, ry=0.000, rz=-0.000, shoulder=lefty, elbow=epositive, wrist=wpositive, fatherId=fReference[0]}
  [253] = {x=-21.302, y=0.000, z=-1.898, rx=-0.000, ry=0.000, rz=-0.000, shoulder=lefty, elbow=epositive, wrist=wpositive, fatherId=fReference[0]}
  [254] = {x=-21.800, y=0.000, z=-1.907, rx=-0.000, ry=0.000, rz=-0.000, shoulder=lefty, elbow=epositive, wrist=wpositive, fatherId=fReference[0]}
  [255] = {x=-22.297, y=0.000, z=-1.915, rx=-0.000, ry=0.000, rz=-0.000, shoulder=lefty, elbow=epositive, wrist=wpositive, fatherId=fReference[0]}
  [256] = {x=-22.794, y=0.000, z=-1.923, rx=-0.000, ry=0.000, rz=-0.000, shoulder=lefty, elbow=epositive, wrist=wpositive, fatherId=fReference[0]}
  [257] = {x=-23.292, y=0.000, z=-1.932, rx=-0.000, ry=0.000, rz=-0.000, shoulder=lefty, elbow=epositive, wrist=wpositive, fatherId=fReference[0]}
  [258] = {x=-23.789, y=0.000, z=-1.940, rx=-0.000, ry=0.000, rz=-0.000, shoulder=lefty, elbow=epositive, wrist=wpositive, fatherId=fReference[0]}
  [259] = {x=-24.287, y=0.000, z=-1.948, rx=-0.000, ry=0.000, rz=-0.000, shoulder=lefty, elbow=epositive, wrist=wpositive, fatherId=fReference[0]}
  [260] = {x=-24.784, y=0.000, z=-1.957, rx=-0.000, ry=0.000, rz=-0.000, shoulder=lefty, elbow=epositive, wrist=wpositive, fatherId=fReference[0]}
  [261] = {x=-25.281, y=0.000, z=-1.965, rx=-0.000, ry=0.000, rz=-0.000, shoulder=lefty, elbow=epositive, wrist=wpositive, fatherId=fReference[0]}
  [262] = {x=-25.778, y=0.000, z=-1.974, rx=-0.000, ry=0.000, rz=-0.000, shoulder=lefty, elbow=epositive, wrist=wpositive, fatherId=fReference[0]}
  [263] = {x=-26.275, y=0.000, z=-1.982, rx=-0.000, ry=0.000, rz=-0.000, shoulder=lefty, elbow=epositive, wrist=wpositive, fatherId=fReference[0]}
  [264] = {x=-26.772, y=0.000, z=-1.991, rx=-0.000, ry=0.000, rz=-0.000, shoulder=lefty, elbow=epositive, wrist=wpositive, fatherId=fReference[0]}
  [265] = {x=-27.269, y=0.000, z=-2.000, rx=-0.000, ry=0.000, rz=-0.000, shoulder=lefty, elbow=epositive, wrist=wpositive, fatherId=fReference[0]}
  [266] = {x=-27.766, y=0.000, z=-2.008, rx=-0.000, ry=0.000, rz=-0.000, shoulder=lefty, elbow=epositive, wrist=wpositive, fatherId=fReference[0]}
  [267] = {x=-28.263, y=0.000, z=-2.017, rx=-0.000, ry=0.000, rz=-0.000, shoulder=lefty, elbow=epositive, wrist=wpositive, fatherId=fReference[0]}
  [268] = {x=-28.760, y=0.000, z=-2.026, rx=-0.000, ry=0.000, rz=-0.000, shoulder=lefty, elbow=epositive, wrist=wpositive, fatherId=fReference[0]}
  [269] = {x=-29.257, y=0.000, z=-2.035, rx=-0.000, ry=0.000, rz=-0.000, shoulder=lefty, elbow=epositive, wrist=wpositive, fatherId=fReference[0]}
  [270] = {x=-29.753, y=0.000, z=-2.043, rx=-0.000, ry=0.000, rz=-0.000, shoulder=lefty, elbow=epositive, wrist=wpositive, fatherId=fReference[0]}
  [271] = {x=-30.250, y=0.000, z=-2.052, rx=-0.000, ry=0.000, rz=-0.000, shoulder=lefty, elbow=epositive, wrist=wpositive, fatherId=fReference[0]}
  [272] = {x=-30.746, y=0.000, z=-2.061, rx=-0.000, ry=0.000, rz=-0.000, shoulder=lefty, elbow=epositive, wrist=wpositive, fatherId=fReference[0]}
  [273] = {x=-31.242, y=0.000, z=-2.070, rx=-0.000, ry=0.000, rz=-0.000, shoulder=lefty, elbow=epositive, wrist=wpositive, fatherId=fReference[0]}
  [274] = {x=-31.739, y=0.000, z=-2.079, rx=-0.000, ry=0.000, rz=-0.000, shoulder=lefty, elbow=epositive, wrist=wpositive, fatherId=fReference[0]}
  [275] = {x=-32.236, y=0.000, z=-2.088, rx=-0.000, ry=0.000, rz=-0.000, shoulder=lefty, elbow=epositive, wrist=wpositive, fatherId=fReference[0]}
  [276] = {x=-32.733, y=0.000, z=-2.097, rx=-0.000, ry=0.000, rz=-0.000, shoulder=lefty, elbow=epositive, wrist=wpositive, fatherId=fReference[0]}
  [277] = {x=-33.229, y=0.000, z=-2.106, rx=-0.000, ry=0.000, rz=-0.000, shoulder=lefty, elbow=epositive, wrist=wpositive, fatherId=fReference[0]}
  [278] = {x=-33.726, y=0.000, z=-2.115, rx=-0.000, ry=0.000, rz=-0.000, shoulder=lefty, elbow=epositive, wrist=wpositive, fatherId=fReference[0]}
  [279] = {x=-33.164, y=0.000, z=-2.113, rx=-0.000, ry=0.000, rz=-0.000, shoulder=lefty, elbow=epositive, wrist=wpositive, fatherId=fReference[0]}
  [280] = {x=-32.669, y=0.000, z=-2.118, rx=-0.000, ry=0.000, rz=-0.000, shoulder=lefty, elbow=epositive, wrist=wpositive, fatherId=fReference[0]}
  [281] = {x=-32.173, y=0.000, z=-2.123, rx=-0.000, ry=0.000, rz=-0.000, shoulder=lefty, elbow=epositive, wrist=wpositive, fatherId=fReference[0]}
  [282] = {x=-31.677, y=0.000, z=-2.129, rx=-0.000, ry=0.000, rz=-0.000, shoulder=lefty, elbow=epositive, wrist=wpositive, fatherId=fReference[0]}
  [283] = {x=-31.180, y=0.000, z=-2.135, rx=-0.000, ry=0.000, rz=-0.000, shoulder=lefty, elbow=epositive, wrist=wpositive, fatherId=fReference[0]}
  [284] = {x=-30.682, y=0.000, z=-2.141, rx=-0.000, ry=0.000, rz=-0.000, shoulder=lefty, elbow=epositive, wrist=wpositive, fatherId=fReference[0]}
  [285] = {x=-30.184, y=0.000, z=-2.148, rx=-0.000, ry=0.000, rz=-0.000, shoulder=lefty, elbow=epositive, wrist=wpositive, fatherId=fReference[0]}
  [286] = {x=-29.686, y=0.000, z=-2.154, rx=-0.000, ry=0.000, rz=-0.000, shoulder=lefty, elbow=epositive, wrist=wpositive, fatherId=fReference[0]}
  [287] = {x=-29.187, y=0.000, z=-2.161, rx=-0.000, ry=0.000, rz=-0.000, shoulder=lefty, elbow=epositive, wrist=wpositive, fatherId=fReference[0]}
  [288] = {x=-28.689, y=0.000, z=-2.168, rx=-0.000, ry=0.000, rz=-0.000, shoulder=lefty, elbow=epositive, wrist=wpositive, fatherId=fReference[0]}
  [289] = {x=-28.189, y=0.000, z=-2.175, rx=-0.000, ry=0.000, rz=-0.000, shoulder=lefty, elbow=epositive, wrist=wpositive, fatherId=fReference[0]}
  [290] = {x=-27.690, y=0.000, z=-2.181, rx=-0.000, ry=0.000, rz=-0.000, shoulder=lefty, elbow=epositive, wrist=wpositive, fatherId=fReference[0]}
  [291] = {x=-27.191, y=0.000, z=-2.188, rx=-0.000, ry=0.000, rz=-0.000, shoulder=lefty, elbow=epositive, wrist=wpositive, fatherId=fReference[0]}
  [292] = {x=-26.692, y=0.000, z=-2.195, rx=-0.000, ry=0.000, rz=-0.000, shoulder=lefty, elbow=epositive, wrist=wpositive, fatherId=fReference[0]}
  [293] = {x=-26.192, y=0.000, z=-2.203, rx=-0.000, ry=0.000, rz=-0.000, shoulder=lefty, elbow=epositive, wrist=wpositive, fatherId=fReference[0]}
  [294] = {x=-25.692, y=0.000, z=-2.210, rx=-0.000, ry=0.000, rz=-0.000, shoulder=lefty, elbow=epositive, wrist=wpositive, fatherId=fReference[0]}
  [295] = {x=-25.192, y=0.000, z=-2.217, rx=-0.000, ry=0.000, rz=-0.000, shoulder=lefty, elbow=epositive, wrist=wpositive, fatherId=fReference[0]}
  [296] = {x=-24.693, y=0.000, z=-2.224, rx=-0.000, ry=0.000, rz=-0.000, shoulder=lefty, elbow=epositive, wrist=wpositive, fatherId=fReference[0]}
  [297] = {x=-24.193, y=0.000, z=-2.231, rx=-0.000, ry=0.000, rz=-0.000, shoulder=lefty, elbow=epositive, wrist=wpositive, fatherId=fReference[0]}
  [298] = {x=-23.693, y=0.000, z=-2.238, rx=-0.000, ry=0.000, rz=-0.000, shoulder=lefty, elbow=epositive, wrist=wpositive, fatherId=fReference[0]}
  [299] = {x=-23.193, y=0.000, z=-2.246, rx=-0.000, ry=0.000, rz=-0.000, shoulder=lefty, elbow=epositive, wrist=wpositive, fatherId=fReference[0]}
  [300] = {x=-22.693, y=0.000, z=-2.253, rx=-0.000, ry=0.000, rz=-0.000, shoulder=lefty, elbow=epositive, wrist=wpositive, fatherId=fReference[0]}
  [301] = {x=-22.193, y=0.000, z=-2.260, rx=-0.000, ry=0.000, rz=-0.000, shoulder=lefty, elbow=epositive, wrist=wpositive, fatherId=fReference[0]}
  [302] = {x=-21.692, y=0.000, z=-2.268, rx=-0.000, ry=0.000, rz=-0.000, shoulder=lefty, elbow=epositive, wrist=wpositive, fatherId=fReference[0]}
  [303] = {x=-21.192, y=0.000, z=-2.275, rx=-0.000, ry=0.000, rz=-0.000, shoulder=lefty, elbow=epositive, wrist=wpositive, fatherId=fReference[0]}
  [304] = {x=-20.692, y=0.000, z=-2.282, rx=-0.000, ry=0.000, rz=-0.000, shoulder=lefty, elbow=epositive, wrist=wpositive, fatherId=fReference[0]}
  [305] = {x=-20.192, y=0.000, z=-2.290, rx=-0.000, ry=0.000, rz=-0.000, shoulder=lefty, elbow=epositive, wrist=wpositive, fatherId=fReference[0]}
  [306] = {x=-19.691, y=0.000, z=-2.297, rx=-0.000, ry=0.000, rz=-0.000, shoulder=lefty, elbow=epositive, wrist=wpositive, fatherId=fReference[0]}
  [307] = {x=-19.191, y=0.000, z=-2.304, rx=-0.000, ry=0.000, rz=-0.000, shoulder=lefty, elbow=epositive, wrist=wpositive, fatherId=fReference[0]}
  [308] = {x=-18.690, y=0.000, z=-2.312, rx=-0.000, ry=0.000, rz=-0.000, shoulder=lefty, elbow=epositive, wrist=wpositive, fatherId=fReference[0]}
  [309] = {x=-18.190, y=0.000, z=-2.319, rx=-0.000, ry=0.000, rz=-0.000, shoulder=lefty, elbow=epositive, wrist=wpositive, fatherId=fReference[0]}
  [310] = {x=-17.689, y=0.000, z=-2.327, rx=-0.000, ry=0.000, rz=-0.000, shoulder=lefty, elbow=epositive, wrist=wpositive, fatherId=fReference[0]}
  [311] = {x=-17.189, y=0.000, z=-2.334, rx=-0.000, ry=0.000, rz=-0.000, shoulder=lefty, elbow=epositive, wrist=wpositive, fatherId=fReference[0]}
  [312] = {x=-16.688, y=0.000, z=-2.342, rx=-0.000, ry=0.000, rz=-0.000, shoulder=lefty, elbow=epositive, wrist=wpositive, fatherId=fReference[0]}
  [313] = {x=-16.188, y=0.000, z=-2.349, rx=-0.000, ry=0.000, rz=-0.000, shoulder=lefty, elbow=epositive, wrist=wpositive, fatherId=fReference[0]}
  [314] = {x=-15.687, y=0.000, z=-2.357, rx=-0.000, ry=0.000, rz=-0.000, shoulder=lefty, elbow=epositive, wrist=wpositive, fatherId=fReference[0]}
  [315] = {x=-15.186, y=0.000, z=-2.364, rx=-0.000, ry=0.000, rz=-0.000, shoulder=lefty, elbow=epositive, wrist=wpositive, fatherId=fReference[0]}
  [316] = {x=-14.685, y=0.000, z=-2.372, rx=-0.000, ry=0.000, rz=-0.000, shoulder=lefty, elbow=epositive, wrist=wpositive, fatherId=fReference[0]}
  [317] = {x=-14.184, y=0.000, z=-2.379, rx=-0.000, ry=0.000, rz=-0.000, shoulder=lefty, elbow=epositive, wrist=wpositive, fatherId=fReference[0]}
  [318] = {x=-13.683, y=0.000, z=-2.387, rx=-0.000, ry=0.000, rz=-0.000, shoulder=lefty, elbow=epositive, wrist=wpositive, fatherId=fReference[0]}
  [319] = {x=-13.182, y=0.000, z=-2.394, rx=-0.000, ry=0.000, rz=-0.000, shoulder=lefty, elbow=epositive, wrist=wpositive, fatherId=fReference[0]}
  [320] = {x=-12.682, y=0.000, z=-2.402, rx=-0.000, ry=0.000, rz=-0.000, shoulder=lefty, elbow=epositive, wrist=wpositive, fatherId=fReference[0]}
  [321] = {x=-12.181, y=0.000, z=-2.409, rx=-0.000, ry=0.000, rz=-0.000, shoulder=lefty, elbow=epositive, wrist=wpositive, fatherId=fReference[0]}
  [322] = {x=-11.680, y=0.000, z=-2.417, rx=-0.000, ry=0.000, rz=-0.000, shoulder=lefty, elbow=epositive, wrist=wpositive, fatherId=fReference[0]}
  [323] = {x=-11.179, y=0.000, z=-2.424, rx=-0.000, ry=0.000, rz=-0.000, shoulder=lefty, elbow=epositive, wrist=wpositive, fatherId=fReference[0]}
  [324] = {x=-10.678, y=0.000, z=-2.432, rx=-0.000, ry=0.000, rz=-0.000, shoulder=lefty, elbow=epositive, wrist=wpositive, fatherId=fReference[0]}
  [325] = {x=-10.177, y=0.000, z=-2.439, rx=-0.000, ry=0.000, rz=-0.000, shoulder=lefty, elbow=epositive, wrist=wpositive, fatherId=fReference[0]}
  [326] = {x=-9.676, y=0.000, z=-2.447, rx=-0.000, ry=0.000, rz=-0.000, shoulder=lefty, elbow=epositive, wrist=wpositive, fatherId=fReference[0]}
  [327] = {x=-9.175, y=0.000, z=-2.454, rx=-0.000, ry=0.000, rz=-0.000, shoulder=lefty, elbow=epositive, wrist=wpositive, fatherId=fReference[0]}
  [328] = {x=-8.674, y=0.000, z=-2.462, rx=-0.000, ry=0.000, rz=-0.000, shoulder=lefty, elbow=epositive, wrist=wpositive, fatherId=fReference[0]}
  [329] = {x=-8.172, y=0.000, z=-2.470, rx=-0.000, ry=0.000, rz=-0.000, shoulder=lefty, elbow=epositive, wrist=wpositive, fatherId=fReference[0]}
  [330] = {x=-7.671, y=0.000, z=-2.477, rx=-0.000, ry=0.000, rz=-0.000, shoulder=lefty, elbow=epositive, wrist=wpositive, fatherId=fReference[0]}
  [331] = {x=-7.170, y=0.000, z=-2.485, rx=-0.000, ry=0.000, rz=-0.000, shoulder=lefty, elbow=epositive, wrist=wpositive, fatherId=fReference[0]}
  [332] = {x=-6.669, y=0.000, z=-2.492, rx=-0.000, ry=0.000, rz=-0.000, shoulder=lefty, elbow=epositive, wrist=wpositive, fatherId=fReference[0]}
  [333] = {x=-6.168, y=0.000, z=-2.500, rx=-0.000, ry=0.000, rz=-0.000, shoulder=lefty, elbow=epositive, wrist=wpositive, fatherId=fReference[0]}
  [334] = {x=-5.666, y=0.000, z=-2.507, rx=-0.000, ry=0.000, rz=-0.000, shoulder=lefty, elbow=epositive, wrist=wpositive, fatherId=fReference[0]}
  [335] = {x=-5.165, y=0.000, z=-2.515, rx=-0.000, ry=0.000, rz=-0.000, shoulder=lefty, elbow=epositive, wrist=wpositive, fatherId=fReference[0]}
  [336] = {x=-4.664, y=0.000, z=-2.523, rx=-0.000, ry=0.000, rz=-0.000, shoulder=lefty, elbow=epositive, wrist=wpositive, fatherId=fReference[0]}
  [337] = {x=-4.162, y=0.000, z=-2.530, rx=-0.000, ry=0.000, rz=-0.000, shoulder=lefty, elbow=epositive, wrist=wpositive, fatherId=fReference[0]}
  [338] = {x=-3.661, y=0.000, z=-2.538, rx=-0.000, ry=0.000, rz=-0.000, shoulder=lefty, elbow=epositive, wrist=wpositive, fatherId=fReference[0]}
  [339] = {x=-3.159, y=0.000, z=-2.546, rx=-0.000, ry=0.000, rz=-0.000, shoulder=lefty, elbow=epositive, wrist=wpositive, fatherId=fReference[0]}
  [340] = {x=-2.658, y=0.000, z=-2.554, rx=-0.000, ry=0.000, rz=-0.000, shoulder=lefty, elbow=epositive, wrist=wpositive, fatherId=fReference[0]}
  [341] = {x=-2.156, y=0.000, z=-2.561, rx=-0.000, ry=0.000, rz=-0.000, shoulder=lefty, elbow=epositive, wrist=wpositive, fatherId=fReference[0]}
  [342] = {x=-1.654, y=0.000, z=-2.569, rx=-0.000, ry=0.000, rz=-0.000, shoulder=lefty, elbow=epositive, wrist=wpositive, fatherId=fReference[0]}
  [343] = {x=-1.153, y=0.000, z=-2.577, rx=-0.000, ry=0.000, rz=-0.000, shoulder=lefty, elbow=epositive, wrist=wpositive, fatherId=fReference[0]}
  [344] = {x=-0.651, y=0.000, z=-2.585, rx=-0.000, ry=0.000, rz=-0.000, shoulder=lefty, elbow=epositive, wrist=wpositive, fatherId=fReference[0]}
  [345] = {x=-0.149, y=0.000, z=-2.592, rx=-0.000, ry=0.000, rz=-0.000, shoulder=lefty, elbow=epositive, wrist=wpositive, fatherId=fReference[0]}
  [346] = {x=0.353, y=0.000, z=-2.600, rx=-0.000, ry=0.000, rz=-0.000, shoulder=lefty, elbow=epositive, wrist=wpositive, fatherId=fReference[0]}
  [347] = {x=0.855, y=0.000, z=-2.608, rx=-0.000, ry=0.000, rz=-0.000, shoulder=lefty, elbow=epositive, wrist=wpositive, fatherId=fReference[0]}
  [348] = {x=1.357, y=0.000, z=-2.616, rx=-0.000, ry=0.000, rz=-0.000, shoulder=lefty, elbow=epositive, wrist=wpositive, fatherId=fReference[0]}
  [349] = {x=1.860, y=0.000, z=-2.624, rx=-0.000, ry=0.000, rz=-0.000, shoulder=lefty, elbow=epositive, wrist=wpositive, fatherId=fReference[0]}
  [350] = {x=2.362, y=0.000, z=-2.632, rx=-0.000, ry=0.000, rz=-0.000, shoulder=lefty, elbow=epositive, wrist=wpositive, fatherId=fReference[0]}
  [351] = {x=2.865, y=0.000, z=-2.640, rx=-0.000, ry=0.000, rz=-0.000, shoulder=lefty, elbow=epositive, wrist=wpositive, fatherId=fReference[0]}
  [352] = {x=3.367, y=0.000, z=-2.648, rx=-0.000, ry=0.000, rz=-0.000, shoulder=lefty, elbow=epositive, wrist=wpositive, fatherId=fReference[0]}
  [353] = {x=3.870, y=0.000, z=-2.656, rx=-0.000, ry=0.000, rz=-0.000, shoulder=lefty, elbow=epositive, wrist=wpositive, fatherId=fReference[0]}
  [354] = {x=4.373, y=0.000, z=-2.664, rx=-0.000, ry=0.000, rz=-0.000, shoulder=lefty, elbow=epositive, wrist=wpositive, fatherId=fReference[0]}
  [355] = {x=4.875, y=0.000, z=-2.672, rx=-0.000, ry=0.000, rz=-0.000, shoulder=lefty, elbow=epositive, wrist=wpositive, fatherId=fReference[0]}
  [356] = {x=5.378, y=0.000, z=-2.680, rx=-0.000, ry=0.000, rz=-0.000, shoulder=lefty, elbow=epositive, wrist=wpositive, fatherId=fReference[0]}
  [357] = {x=5.881, y=0.000, z=-2.688, rx=-0.000, ry=0.000, rz=-0.000, shoulder=lefty, elbow=epositive, wrist=wpositive, fatherId=fReference[0]}
  [358] = {x=6.383, y=0.000, z=-2.696, rx=-0.000, ry=0.000, rz=-0.000, shoulder=lefty, elbow=epositive, wrist=wpositive, fatherId=fReference[0]}
  [359] = {x=6.886, y=0.000, z=-2.704, rx=-0.000, ry=0.000, rz=-0.000, shoulder=lefty, elbow=epositive, wrist=wpositive, fatherId=fReference[0]}
  [360] = {x=7.389, y=0.000, z=-2.712, rx=-0.000, ry=0.000, rz=-0.000, shoulder=lefty, elbow=epositive, wrist=wpositive, fatherId=fReference[0]}
  [361] = {x=7.892, y=0.000, z=-2.720, rx=-0.000, ry=0.000, rz=-0.000, shoulder=lefty, elbow=epositive, wrist=wpositive, fatherId=fReference[0]}
  [362] = {x=8.396, y=0.000, z=-2.728, rx=-0.000, ry=0.000, rz=-0.000, shoulder=lefty, elbow=epositive, wrist=wpositive, fatherId=fReference[0]}
  [363] = {x=8.899, y=0.000, z=-2.736, rx=-0.000, ry=0.000, rz=-0.000, shoulder=lefty, elbow=epositive, wrist=wpositive, fatherId=fReference[0]}
  [364] = {x=9.402, y=0.000, z=-2.745, rx=-0.000, ry=0.000, rz=-0.000, shoulder=lefty, elbow=epositive, wrist=wpositive, fatherId=fReference[0]}
  [365] = {x=9.905, y=0.000, z=-2.753, rx=-0.000, ry=0.000, rz=-0.000, shoulder=lefty, elbow=epositive, wrist=wpositive, fatherId=fReference[0]}
  [366] = {x=10.409, y=0.000, z=-2.761, rx=-0.000, ry=0.000, rz=-0.000, shoulder=lefty, elbow=epositive, wrist=wpositive, fatherId=fReference[0]}
  [367] = {x=10.912, y=0.000, z=-2.769, rx=-0.000, ry=0.000, rz=-0.000, shoulder=lefty, elbow=epositive, wrist=wpositive, fatherId=fReference[0]}
  [368] = {x=11.415, y=0.000, z=-2.777, rx=-0.000, ry=0.000, rz=-0.000, shoulder=lefty, elbow=epositive, wrist=wpositive, fatherId=fReference[0]}
  [369] = {x=11.919, y=0.000, z=-2.786, rx=-0.000, ry=0.000, rz=-0.000, shoulder=lefty, elbow=epositive, wrist=wpositive, fatherId=fReference[0]}
  [370] = {x=12.422, y=0.000, z=-2.794, rx=-0.000, ry=0.000, rz=-0.000, shoulder=lefty, elbow=epositive, wrist=wpositive, fatherId=fReference[0]}
  [371] = {x=12.926, y=0.000, z=-2.802, rx=-0.000, ry=0.000, rz=-0.000, shoulder=lefty, elbow=epositive, wrist=wpositive, fatherId=fReference[0]}
  [372] = {x=13.430, y=0.000, z=-2.810, rx=-0.000, ry=0.000, rz=-0.000, shoulder=lefty, elbow=epositive, wrist=wpositive, fatherId=fReference[0]}
  [373] = {x=13.934, y=0.000, z=-2.819, rx=-0.000, ry=0.000, rz=-0.000, shoulder=lefty, elbow=epositive, wrist=wpositive, fatherId=fReference[0]}
  [374] = {x=14.437, y=0.000, z=-2.827, rx=-0.000, ry=0.000, rz=-0.000, shoulder=lefty, elbow=epositive, wrist=wpositive, fatherId=fReference[0]}
  [375] = {x=14.941, y=0.000, z=-2.835, rx=-0.000, ry=0.000, rz=-0.000, shoulder=lefty, elbow=epositive, wrist=wpositive, fatherId=fReference[0]}
  [376] = {x=15.445, y=0.000, z=-2.843, rx=-0.000, ry=0.000, rz=-0.000, shoulder=lefty, elbow=epositive, wrist=wpositive, fatherId=fReference[0]}
  [377] = {x=15.950, y=0.000, z=-2.852, rx=-0.000, ry=0.000, rz=-0.000, shoulder=lefty, elbow=epositive, wrist=wpositive, fatherId=fReference[0]}
  [378] = {x=16.454, y=0.000, z=-2.860, rx=-0.000, ry=0.000, rz=-0.000, shoulder=lefty, elbow=epositive, wrist=wpositive, fatherId=fReference[0]}
  [379] = {x=16.958, y=0.000, z=-2.868, rx=-0.000, ry=0.000, rz=-0.000, shoulder=lefty, elbow=epositive, wrist=wpositive, fatherId=fReference[0]}
  [380] = {x=17.462, y=0.000, z=-2.877, rx=-0.000, ry=0.000, rz=-0.000, shoulder=lefty, elbow=epositive, wrist=wpositive, fatherId=fReference[0]}
  [381] = {x=17.967, y=0.000, z=-2.885, rx=-0.000, ry=0.000, rz=-0.000, shoulder=lefty, elbow=epositive, wrist=wpositive, fatherId=fReference[0]}
  [382] = {x=18.471, y=0.000, z=-2.893, rx=-0.000, ry=0.000, rz=-0.000, shoulder=lefty, elbow=epositive, wrist=wpositive, fatherId=fReference[0]}
  [383] = {x=18.976, y=0.000, z=-2.902, rx=-0.000, ry=0.000, rz=-0.000, shoulder=lefty, elbow=epositive, wrist=wpositive, fatherId=fReference[0]}
  [384] = {x=19.480, y=0.000, z=-2.910, rx=-0.000, ry=0.000, rz=-0.000, shoulder=lefty, elbow=epositive, wrist=wpositive, fatherId=fReference[0]}
  [385] = {x=19.985, y=0.000, z=-2.919, rx=-0.000, ry=0.000, rz=-0.000, shoulder=lefty, elbow=epositive, wrist=wpositive, fatherId=fReference[0]}
  [386] = {x=20.490, y=0.000, z=-2.927, rx=-0.000, ry=0.000, rz=-0.000, shoulder=lefty, elbow=epositive, wrist=wpositive, fatherId=fReference[0]}
  [387] = {x=20.995, y=0.000, z=-2.936, rx=-0.000, ry=0.000, rz=-0.000, shoulder=lefty, elbow=epositive, wrist=wpositive, fatherId=fReference[0]}
  [388] = {x=21.500, y=0.000, z=-2.944, rx=-0.000, ry=0.000, rz=-0.000, shoulder=lefty, elbow=epositive, wrist=wpositive, fatherId=fReference[0]}
  [389] = {x=22.005, y=0.000, z=-2.952, rx=-0.000, ry=0.000, rz=-0.000, shoulder=lefty, elbow=epositive, wrist=wpositive, fatherId=fReference[0]}
  [390] = {x=22.511, y=0.000, z=-2.961, rx=-0.000, ry=0.000, rz=-0.000, shoulder=lefty, elbow=epositive, wrist=wpositive, fatherId=fReference[0]}
  [391] = {x=23.016, y=0.000, z=-2.970, rx=-0.000, ry=0.000, rz=-0.000, shoulder=lefty, elbow=epositive, wrist=wpositive, fatherId=fReference[0]}
  [392] = {x=23.522, y=0.000, z=-2.978, rx=-0.000, ry=0.000, rz=-0.000, shoulder=lefty, elbow=epositive, wrist=wpositive, fatherId=fReference[0]}
  [393] = {x=24.027, y=0.000, z=-2.986, rx=-0.000, ry=0.000, rz=-0.000, shoulder=lefty, elbow=epositive, wrist=wpositive, fatherId=fReference[0]}
  [394] = {x=24.533, y=0.000, z=-2.995, rx=-0.000, ry=0.000, rz=-0.000, shoulder=lefty, elbow=epositive, wrist=wpositive, fatherId=fReference[0]}
  [395] = {x=25.039, y=0.000, z=-3.003, rx=-0.000, ry=0.000, rz=-0.000, shoulder=lefty, elbow=epositive, wrist=wpositive, fatherId=fReference[0]}
  [396] = {x=25.544, y=0.000, z=-3.012, rx=-0.000, ry=0.000, rz=-0.000, shoulder=lefty, elbow=epositive, wrist=wpositive, fatherId=fReference[0]}
  [397] = {x=26.050, y=0.000, z=-3.021, rx=-0.000, ry=0.000, rz=-0.000, shoulder=lefty, elbow=epositive, wrist=wpositive, fatherId=fReference[0]}
  [398] = {x=26.556, y=0.000, z=-3.029, rx=-0.000, ry=0.000, rz=-0.000, shoulder=lefty, elbow=epositive, wrist=wpositive, fatherId=fReference[0]}
  [399] = {x=27.062, y=0.000, z=-3.038, rx=-0.000, ry=0.000, rz=-0.000, shoulder=lefty, elbow=epositive, wrist=wpositive, fatherId=fReference[0]}
  [400] = {x=27.569, y=0.000, z=-3.047, rx=-0.000, ry=0.000, rz=-0.000, shoulder=lefty, elbow=epositive, wrist=wpositive, fatherId=fReference[0]}
  [401] = {x=28.076, y=0.000, z=-3.056, rx=-0.000, ry=0.000, rz=-0.000, shoulder=lefty, elbow=epositive, wrist=wpositive, fatherId=fReference[0]}
  [402] = {x=28.583, y=0.000, z=-3.065, rx=-0.000, ry=0.000, rz=-0.000, shoulder=lefty, elbow=epositive, wrist=wpositive, fatherId=fReference[0]}
  [403] = {x=29.089, y=0.000, z=-3.073, rx=-0.000, ry=0.000, rz=-0.000, shoulder=lefty, elbow=epositive, wrist=wpositive, fatherId=fReference[0]}
  [404] = {x=29.597, y=0.000, z=-3.083, rx=-0.000, ry=0.000, rz=-0.000, shoulder=lefty, elbow=epositive, wrist=wpositive, fatherId=fReference[0]}
  [405] = {x=30.104, y=0.000, z=-3.092, rx=-0.000, ry=0.000, rz=-0.000, shoulder=lefty, elbow=epositive, wrist=wpositive, fatherId=fReference[0]}
  [406] = {x=30.612, y=0.000, z=-3.101, rx=-0.000, ry=0.000, rz=-0.000, shoulder=lefty, elbow=epositive, wrist=wpositive, fatherId=fReference[0]}
  [407] = {x=31.120, y=0.000, z=-3.110, rx=-0.000, ry=0.000, rz=-0.000, shoulder=lefty, elbow=epositive, wrist=wpositive, fatherId=fReference[0]}
  [408] = {x=31.628, y=0.000, z=-3.119, rx=-0.000, ry=0.000, rz=-0.000, shoulder=lefty, elbow=epositive, wrist=wpositive, fatherId=fReference[0]}
  [409] = {x=32.137, y=0.000, z=-3.128, rx=-0.000, ry=0.000, rz=-0.000, shoulder=lefty, elbow=epositive, wrist=wpositive, fatherId=fReference[0]}
  [410] = {x=32.646, y=0.000, z=-3.137, rx=-0.000, ry=0.000, rz=-0.000, shoulder=lefty, elbow=epositive, wrist=wpositive, fatherId=fReference[0]}
  [411] = {x=33.155, y=0.000, z=-3.147, rx=-0.000, ry=0.000, rz=-0.000, shoulder=lefty, elbow=epositive, wrist=wpositive, fatherId=fReference[0]}
  [412] = {x=33.665, y=0.000, z=-3.156, rx=-0.000, ry=0.000, rz=-0.000, shoulder=lefty, elbow=epositive, wrist=wpositive, fatherId=fReference[0]}
  [413] = {x=34.175, y=0.000, z=-3.166, rx=-0.000, ry=0.000, rz=-0.000, shoulder=lefty, elbow=epositive, wrist=wpositive, fatherId=fReference[0]}
  [414] = {x=34.686, y=0.000, z=-3.175, rx=-0.000, ry=0.000, rz=-0.000, shoulder=lefty, elbow=epositive, wrist=wpositive, fatherId=fReference[0]}
  [415] = {x=34.030, y=0.000, z=-3.185, rx=-0.000, ry=0.000, rz=-0.000, shoulder=lefty, elbow=epositive, wrist=wpositive, fatherId=fReference[0]}
  [416] = {x=33.495, y=0.000, z=-3.187, rx=-0.000, ry=0.000, rz=-0.000, shoulder=lefty, elbow=epositive, wrist=wpositive, fatherId=fReference[0]}
  [417] = {x=32.972, y=0.000, z=-3.190, rx=-0.000, ry=0.000, rz=-0.000, shoulder=lefty, elbow=epositive, wrist=wpositive, fatherId=fReference[0]}
  [418] = {x=32.456, y=0.000, z=-3.195, rx=-0.000, ry=0.000, rz=-0.000, shoulder=lefty, elbow=epositive, wrist=wpositive, fatherId=fReference[0]}
  [419] = {x=31.944, y=0.000, z=-3.200, rx=-0.000, ry=0.000, rz=-0.000, shoulder=lefty, elbow=epositive, wrist=wpositive, fatherId=fReference[0]}
  [420] = {x=31.436, y=0.000, z=-3.206, rx=-0.000, ry=0.000, rz=-0.000, shoulder=lefty, elbow=epositive, wrist=wpositive, fatherId=fReference[0]}
  [421] = {x=30.930, y=0.000, z=-3.212, rx=-0.000, ry=0.000, rz=-0.000, shoulder=lefty, elbow=epositive, wrist=wpositive, fatherId=fReference[0]}
  [422] = {x=30.427, y=0.000, z=-3.219, rx=-0.000, ry=0.000, rz=-0.000, shoulder=lefty, elbow=epositive, wrist=wpositive, fatherId=fReference[0]}
  [423] = {x=29.925, y=0.000, z=-3.226, rx=-0.000, ry=0.000, rz=-0.000, shoulder=lefty, elbow=epositive, wrist=wpositive, fatherId=fReference[0]}
  [424] = {x=29.423, y=0.000, z=-3.234, rx=-0.000, ry=0.000, rz=-0.000, shoulder=lefty, elbow=epositive, wrist=wpositive, fatherId=fReference[0]}
  [425] = {x=28.921, y=0.000, z=-3.241, rx=-0.000, ry=0.000, rz=-0.000, shoulder=lefty, elbow=epositive, wrist=wpositive, fatherId=fReference[0]}
  [426] = {x=28.421, y=0.000, z=-3.249, rx=-0.000, ry=0.000, rz=-0.000, shoulder=lefty, elbow=epositive, wrist=wpositive, fatherId=fReference[0]}
  [427] = {x=27.921, y=0.000, z=-3.257, rx=-0.000, ry=0.000, rz=-0.000, shoulder=lefty, elbow=epositive, wrist=wpositive, fatherId=fReference[0]}
  [428] = {x=27.421, y=0.000, z=-3.264, rx=-0.000, ry=0.000, rz=-0.000, shoulder=lefty, elbow=epositive, wrist=wpositive, fatherId=fReference[0]}
  [429] = {x=26.921, y=0.000, z=-3.272, rx=-0.000, ry=0.000, rz=-0.000, shoulder=lefty, elbow=epositive, wrist=wpositive, fatherId=fReference[0]}
  [430] = {x=26.422, y=0.000, z=-3.280, rx=-0.000, ry=0.000, rz=-0.000, shoulder=lefty, elbow=epositive, wrist=wpositive, fatherId=fReference[0]}
  [431] = {x=25.923, y=0.000, z=-3.288, rx=-0.000, ry=0.000, rz=-0.000, shoulder=lefty, elbow=epositive, wrist=wpositive, fatherId=fReference[0]}
  [432] = {x=25.424, y=0.000, z=-3.296, rx=-0.000, ry=0.000, rz=-0.000, shoulder=lefty, elbow=epositive, wrist=wpositive, fatherId=fReference[0]}
  [433] = {x=24.926, y=0.000, z=-3.305, rx=-0.000, ry=0.000, rz=-0.000, shoulder=lefty, elbow=epositive, wrist=wpositive, fatherId=fReference[0]}
  [434] = {x=24.428, y=0.000, z=-3.313, rx=-0.000, ry=0.000, rz=-0.000, shoulder=lefty, elbow=epositive, wrist=wpositive, fatherId=fReference[0]}
  [435] = {x=23.929, y=0.000, z=-3.321, rx=-0.000, ry=0.000, rz=-0.000, shoulder=lefty, elbow=epositive, wrist=wpositive, fatherId=fReference[0]}
  [436] = {x=23.431, y=0.000, z=-3.329, rx=-0.000, ry=0.000, rz=-0.000, shoulder=lefty, elbow=epositive, wrist=wpositive, fatherId=fReference[0]}
  [437] = {x=22.933, y=0.000, z=-3.338, rx=-0.000, ry=0.000, rz=-0.000, shoulder=lefty, elbow=epositive, wrist=wpositive, fatherId=fReference[0]}
  [438] = {x=22.434, y=0.000, z=-3.346, rx=-0.000, ry=0.000, rz=-0.000, shoulder=lefty, elbow=epositive, wrist=wpositive, fatherId=fReference[0]}
  [439] = {x=21.936, y=0.000, z=-3.354, rx=-0.000, ry=0.000, rz=-0.000, shoulder=lefty, elbow=epositive, wrist=wpositive, fatherId=fReference[0]}
  [440] = {x=21.437, y=0.000, z=-3.362, rx=-0.000, ry=0.000, rz=-0.000, shoulder=lefty, elbow=epositive, wrist=wpositive, fatherId=fReference[0]}
  [441] = {x=20.938, y=0.000, z=-3.370, rx=-0.000, ry=0.000, rz=-0.000, shoulder=lefty, elbow=epositive, wrist=wpositive, fatherId=fReference[0]}
  [442] = {x=20.439, y=0.000, z=-3.378, rx=-0.000, ry=0.000, rz=-0.000, shoulder=lefty, elbow=epositive, wrist=wpositive, fatherId=fReference[0]}
  [443] = {x=19.940, y=0.000, z=-3.386, rx=-0.000, ry=0.000, rz=-0.000, shoulder=lefty, elbow=epositive, wrist=wpositive, fatherId=fReference[0]}
  [444] = {x=19.441, y=0.000, z=-3.394, rx=-0.000, ry=0.000, rz=-0.000, shoulder=lefty, elbow=epositive, wrist=wpositive, fatherId=fReference[0]}
  [445] = {x=18.941, y=0.000, z=-3.402, rx=-0.000, ry=0.000, rz=-0.000, shoulder=lefty, elbow=epositive, wrist=wpositive, fatherId=fReference[0]}
  [446] = {x=18.442, y=0.000, z=-3.410, rx=-0.000, ry=0.000, rz=-0.000, shoulder=lefty, elbow=epositive, wrist=wpositive, fatherId=fReference[0]}
  [447] = {x=17.943, y=0.000, z=-3.418, rx=-0.000, ry=0.000, rz=-0.000, shoulder=lefty, elbow=epositive, wrist=wpositive, fatherId=fReference[0]}
  [448] = {x=17.443, y=0.000, z=-3.426, rx=-0.000, ry=0.000, rz=-0.000, shoulder=lefty, elbow=epositive, wrist=wpositive, fatherId=fReference[0]}
  [449] = {x=16.944, y=0.000, z=-3.434, rx=-0.000, ry=0.000, rz=-0.000, shoulder=lefty, elbow=epositive, wrist=wpositive, fatherId=fReference[0]}
  [450] = {x=16.444, y=0.000, z=-3.442, rx=-0.000, ry=0.000, rz=-0.000, shoulder=lefty, elbow=epositive, wrist=wpositive, fatherId=fReference[0]}
  [451] = {x=15.944, y=0.000, z=-3.449, rx=-0.000, ry=0.000, rz=-0.000, shoulder=lefty, elbow=epositive, wrist=wpositive, fatherId=fReference[0]}
  [452] = {x=15.445, y=0.000, z=-3.457, rx=-0.000, ry=0.000, rz=-0.000, shoulder=lefty, elbow=epositive, wrist=wpositive, fatherId=fReference[0]}
  [453] = {x=14.945, y=0.000, z=-3.465, rx=-0.000, ry=0.000, rz=-0.000, shoulder=lefty, elbow=epositive, wrist=wpositive, fatherId=fReference[0]}
  [454] = {x=14.445, y=0.000, z=-3.473, rx=-0.000, ry=0.000, rz=-0.000, shoulder=lefty, elbow=epositive, wrist=wpositive, fatherId=fReference[0]}
  [455] = {x=13.945, y=0.000, z=-3.481, rx=-0.000, ry=0.000, rz=-0.000, shoulder=lefty, elbow=epositive, wrist=wpositive, fatherId=fReference[0]}
  [456] = {x=13.445, y=0.000, z=-3.489, rx=-0.000, ry=0.000, rz=-0.000, shoulder=lefty, elbow=epositive, wrist=wpositive, fatherId=fReference[0]}
  [457] = {x=12.945, y=0.000, z=-3.496, rx=-0.000, ry=0.000, rz=-0.000, shoulder=lefty, elbow=epositive, wrist=wpositive, fatherId=fReference[0]}
  [458] = {x=12.445, y=0.000, z=-3.504, rx=-0.000, ry=0.000, rz=-0.000, shoulder=lefty, elbow=epositive, wrist=wpositive, fatherId=fReference[0]}
  [459] = {x=11.945, y=0.000, z=-3.512, rx=-0.000, ry=0.000, rz=-0.000, shoulder=lefty, elbow=epositive, wrist=wpositive, fatherId=fReference[0]}
  [460] = {x=11.445, y=0.000, z=-3.520, rx=-0.000, ry=0.000, rz=-0.000, shoulder=lefty, elbow=epositive, wrist=wpositive, fatherId=fReference[0]}
  [461] = {x=10.945, y=0.000, z=-3.527, rx=-0.000, ry=0.000, rz=-0.000, shoulder=lefty, elbow=epositive, wrist=wpositive, fatherId=fReference[0]}
  [462] = {x=10.445, y=0.000, z=-3.535, rx=-0.000, ry=0.000, rz=-0.000, shoulder=lefty, elbow=epositive, wrist=wpositive, fatherId=fReference[0]}
  [463] = {x=9.945, y=0.000, z=-3.543, rx=-0.000, ry=0.000, rz=-0.000, shoulder=lefty, elbow=epositive, wrist=wpositive, fatherId=fReference[0]}
  [464] = {x=9.445, y=0.000, z=-3.551, rx=-0.000, ry=0.000, rz=-0.000, shoulder=lefty, elbow=epositive, wrist=wpositive, fatherId=fReference[0]}
  [465] = {x=8.946, y=0.000, z=-3.559, rx=-0.000, ry=0.000, rz=-0.000, shoulder=lefty, elbow=epositive, wrist=wpositive, fatherId=fReference[0]}
  [466] = {x=8.446, y=0.000, z=-3.567, rx=-0.000, ry=0.000, rz=-0.000, shoulder=lefty, elbow=epositive, wrist=wpositive, fatherId=fReference[0]}
  [467] = {x=7.946, y=0.000, z=-3.574, rx=-0.000, ry=0.000, rz=-0.000, shoulder=lefty, elbow=epositive, wrist=wpositive, fatherId=fReference[0]}
  [468] = {x=7.447, y=0.000, z=-3.582, rx=-0.000, ry=0.000, rz=-0.000, shoulder=lefty, elbow=epositive, wrist=wpositive, fatherId=fReference[0]}
  [469] = {x=6.947, y=0.000, z=-3.590, rx=-0.000, ry=0.000, rz=-0.000, shoulder=lefty, elbow=epositive, wrist=wpositive, fatherId=fReference[0]}
  [470] = {x=6.448, y=0.000, z=-3.598, rx=-0.000, ry=0.000, rz=-0.000, shoulder=lefty, elbow=epositive, wrist=wpositive, fatherId=fReference[0]}
  [471] = {x=5.948, y=0.000, z=-3.606, rx=-0.000, ry=0.000, rz=-0.000, shoulder=lefty, elbow=epositive, wrist=wpositive, fatherId=fReference[0]}
  [472] = {x=5.449, y=0.000, z=-3.614, rx=-0.000, ry=0.000, rz=-0.000, shoulder=lefty, elbow=epositive, wrist=wpositive, fatherId=fReference[0]}
  [473] = {x=4.949, y=0.000, z=-3.622, rx=-0.000, ry=0.000, rz=-0.000, shoulder=lefty, elbow=epositive, wrist=wpositive, fatherId=fReference[0]}
  [474] = {x=4.450, y=0.000, z=-3.630, rx=-0.000, ry=0.000, rz=-0.000, shoulder=lefty, elbow=epositive, wrist=wpositive, fatherId=fReference[0]}
  [475] = {x=3.951, y=0.000, z=-3.638, rx=-0.000, ry=0.000, rz=-0.000, shoulder=lefty, elbow=epositive, wrist=wpositive, fatherId=fReference[0]}
  [476] = {x=3.451, y=0.000, z=-3.646, rx=-0.000, ry=0.000, rz=-0.000, shoulder=lefty, elbow=epositive, wrist=wpositive, fatherId=fReference[0]}
  [477] = {x=2.952, y=0.000, z=-3.654, rx=-0.000, ry=0.000, rz=-0.000, shoulder=lefty, elbow=epositive, wrist=wpositive, fatherId=fReference[0]}
  [478] = {x=2.453, y=0.000, z=-3.663, rx=-0.000, ry=0.000, rz=-0.000, shoulder=lefty, elbow=epositive, wrist=wpositive, fatherId=fReference[0]}
  [479] = {x=1.954, y=0.000, z=-3.671, rx=-0.000, ry=0.000, rz=-0.000, shoulder=lefty, elbow=epositive, wrist=wpositive, fatherId=fReference[0]}
  [480] = {x=1.455, y=0.000, z=-3.679, rx=-0.000, ry=0.000, rz=-0.000, shoulder=lefty, elbow=epositive, wrist=wpositive, fatherId=fReference[0]}
  [481] = {x=0.956, y=0.000, z=-3.687, rx=-0.000, ry=0.000, rz=-0.000, shoulder=lefty, elbow=epositive, wrist=wpositive, fatherId=fReference[0]}
  [482] = {x=0.457, y=0.000, z=-3.696, rx=-0.000, ry=0.000, rz=-0.000, shoulder=lefty, elbow=epositive, wrist=wpositive, fatherId=fReference[0]}
  [483] = {x=-0.042, y=0.000, z=-3.704, rx=-0.000, ry=0.000, rz=-0.000, shoulder=lefty, elbow=epositive, wrist=wpositive, fatherId=fReference[0]}
  [484] = {x=-0.540, y=0.000, z=-3.712, rx=-0.000, ry=0.000, rz=-0.000, shoulder=lefty, elbow=epositive, wrist=wpositive, fatherId=fReference[0]}
  [485] = {x=-1.039, y=0.000, z=-3.720, rx=-0.000, ry=0.000, rz=-0.000, shoulder=lefty, elbow=epositive, wrist=wpositive, fatherId=fReference[0]}
  [486] = {x=-1.537, y=0.000, z=-3.729, rx=-0.000, ry=0.000, rz=-0.000, shoulder=lefty, elbow=epositive, wrist=wpositive, fatherId=fReference[0]}
  [487] = {x=-2.036, y=0.000, z=-3.737, rx=-0.000, ry=0.000, rz=-0.000, shoulder=lefty, elbow=epositive, wrist=wpositive, fatherId=fReference[0]}
  [488] = {x=-2.534, y=0.000, z=-3.746, rx=-0.000, ry=0.000, rz=-0.000, shoulder=lefty, elbow=epositive, wrist=wpositive, fatherId=fReference[0]}
  [489] = {x=-3.033, y=0.000, z=-3.754, rx=-0.000, ry=0.000, rz=-0.000, shoulder=lefty, elbow=epositive, wrist=wpositive, fatherId=fReference[0]}
  [490] = {x=-3.531, y=0.000, z=-3.763, rx=-0.000, ry=0.000, rz=-0.000, shoulder=lefty, elbow=epositive, wrist=wpositive, fatherId=fReference[0]}
  [491] = {x=-4.030, y=0.000, z=-3.771, rx=-0.000, ry=0.000, rz=-0.000, shoulder=lefty, elbow=epositive, wrist=wpositive, fatherId=fReference[0]}
  [492] = {x=-4.530, y=0.000, z=-3.779, rx=-0.000, ry=0.000, rz=-0.000, shoulder=lefty, elbow=epositive, wrist=wpositive, fatherId=fReference[0]}
  [493] = {x=-5.028, y=0.000, z=-3.788, rx=-0.000, ry=0.000, rz=-0.000, shoulder=lefty, elbow=epositive, wrist=wpositive, fatherId=fReference[0]}
  [494] = {x=-5.526, y=0.000, z=-3.796, rx=-0.000, ry=0.000, rz=-0.000, shoulder=lefty, elbow=epositive, wrist=wpositive, fatherId=fReference[0]}
  [495] = {x=-6.025, y=0.000, z=-3.805, rx=-0.000, ry=0.000, rz=-0.000, shoulder=lefty, elbow=epositive, wrist=wpositive, fatherId=fReference[0]}
  [496] = {x=-6.524, y=0.000, z=-3.813, rx=-0.000, ry=0.000, rz=-0.000, shoulder=lefty, elbow=epositive, wrist=wpositive, fatherId=fReference[0]}
  [497] = {x=-7.022, y=0.000, z=-3.821, rx=-0.000, ry=0.000, rz=-0.000, shoulder=lefty, elbow=epositive, wrist=wpositive, fatherId=fReference[0]}
  [498] = {x=-7.521, y=0.000, z=-3.830, rx=-0.000, ry=0.000, rz=-0.000, shoulder=lefty, elbow=epositive, wrist=wpositive, fatherId=fReference[0]}
  [499] = {x=-8.020, y=0.000, z=-3.838, rx=-0.000, ry=0.000, rz=-0.000, shoulder=lefty, elbow=epositive, wrist=wpositive, fatherId=fReference[0]}
  [500] = {x=-8.520, y=0.000, z=-3.847, rx=-0.000, ry=0.000, rz=-0.000, shoulder=lefty, elbow=epositive, wrist=wpositive, fatherId=fReference[0]}
  [501] = {x=-9.019, y=0.000, z=-3.855, rx=-0.000, ry=0.000, rz=-0.000, shoulder=lefty, elbow=epositive, wrist=wpositive, fatherId=fReference[0]}
  [502] = {x=-9.518, y=0.000, z=-3.864, rx=-0.000, ry=0.000, rz=-0.000, shoulder=lefty, elbow=epositive, wrist=wpositive, fatherId=fReference[0]}
  [503] = {x=-10.017, y=0.000, z=-3.872, rx=-0.000, ry=0.000, rz=-0.000, shoulder=lefty, elbow=epositive, wrist=wpositive, fatherId=fReference[0]}
  [504] = {x=-10.516, y=0.000, z=-3.881, rx=-0.000, ry=0.000, rz=-0.000, shoulder=lefty, elbow=epositive, wrist=wpositive, fatherId=fReference[0]}
  [505] = {x=-11.015, y=0.000, z=-3.889, rx=-0.000, ry=0.000, rz=-0.000, shoulder=lefty, elbow=epositive, wrist=wpositive, fatherId=fReference[0]}
  [506] = {x=-11.515, y=0.000, z=-3.898, rx=-0.000, ry=0.000, rz=-0.000, shoulder=lefty, elbow=epositive, wrist=wpositive, fatherId=fReference[0]}
  [507] = {x=-12.012, y=0.000, z=-3.907, rx=-0.000, ry=0.000, rz=-0.000, shoulder=lefty, elbow=epositive, wrist=wpositive, fatherId=fReference[0]}
  [508] = {x=-12.511, y=0.000, z=-3.915, rx=-0.000, ry=0.000, rz=-0.000, shoulder=lefty, elbow=epositive, wrist=wpositive, fatherId=fReference[0]}
  [509] = {x=-13.010, y=0.000, z=-3.924, rx=-0.000, ry=0.000, rz=-0.000, shoulder=lefty, elbow=epositive, wrist=wpositive, fatherId=fReference[0]}
  [510] = {x=-13.509, y=0.000, z=-3.932, rx=-0.000, ry=0.000, rz=-0.000, shoulder=lefty, elbow=epositive, wrist=wpositive, fatherId=fReference[0]}
  [511] = {x=-14.006, y=0.000, z=-3.941, rx=-0.000, ry=0.000, rz=-0.000, shoulder=lefty, elbow=epositive, wrist=wpositive, fatherId=fReference[0]}
  [512] = {x=-14.503, y=0.000, z=-3.950, rx=-0.000, ry=0.000, rz=-0.000, shoulder=lefty, elbow=epositive, wrist=wpositive, fatherId=fReference[0]}
  [513] = {x=-15.004, y=0.000, z=-3.959, rx=-0.000, ry=0.000, rz=-0.000, shoulder=lefty, elbow=epositive, wrist=wpositive, fatherId=fReference[0]}
  [514] = {x=-15.503, y=0.000, z=-3.967, rx=-0.000, ry=0.000, rz=-0.000, shoulder=lefty, elbow=epositive, wrist=wpositive, fatherId=fReference[0]}
  [515] = {x=-16.001, y=0.000, z=-3.976, rx=-0.000, ry=0.000, rz=-0.000, shoulder=lefty, elbow=epositive, wrist=wpositive, fatherId=fReference[0]}
  [516] = {x=-16.500, y=0.000, z=-3.985, rx=-0.000, ry=0.000, rz=-0.000, shoulder=lefty, elbow=epositive, wrist=wpositive, fatherId=fReference[0]}
  [517] = {x=-16.999, y=0.000, z=-3.994, rx=-0.000, ry=0.000, rz=-0.000, shoulder=lefty, elbow=epositive, wrist=wpositive, fatherId=fReference[0]}
  [518] = {x=-17.497, y=0.000, z=-4.003, rx=-0.000, ry=0.000, rz=-0.000, shoulder=lefty, elbow=epositive, wrist=wpositive, fatherId=fReference[0]}
  [519] = {x=-17.997, y=0.000, z=-4.011, rx=-0.000, ry=0.000, rz=-0.000, shoulder=lefty, elbow=epositive, wrist=wpositive, fatherId=fReference[0]}
  [520] = {x=-18.495, y=0.000, z=-4.020, rx=-0.000, ry=0.000, rz=-0.000, shoulder=lefty, elbow=epositive, wrist=wpositive, fatherId=fReference[0]}
  [521] = {x=-18.993, y=0.000, z=-4.029, rx=-0.000, ry=0.000, rz=-0.000, shoulder=lefty, elbow=epositive, wrist=wpositive, fatherId=fReference[0]}
  [522] = {x=-19.492, y=0.000, z=-4.038, rx=-0.000, ry=0.000, rz=-0.000, shoulder=lefty, elbow=epositive, wrist=wpositive, fatherId=fReference[0]}
  [523] = {x=-19.990, y=0.000, z=-4.047, rx=-0.000, ry=0.000, rz=-0.000, shoulder=lefty, elbow=epositive, wrist=wpositive, fatherId=fReference[0]}
  [524] = {x=-20.488, y=0.000, z=-4.056, rx=-0.000, ry=0.000, rz=-0.000, shoulder=lefty, elbow=epositive, wrist=wpositive, fatherId=fReference[0]}
  [525] = {x=-20.986, y=0.000, z=-4.065, rx=-0.000, ry=0.000, rz=-0.000, shoulder=lefty, elbow=epositive, wrist=wpositive, fatherId=fReference[0]}
  [526] = {x=-21.484, y=0.000, z=-4.074, rx=-0.000, ry=0.000, rz=-0.000, shoulder=lefty, elbow=epositive, wrist=wpositive, fatherId=fReference[0]}
  [527] = {x=-21.984, y=0.000, z=-4.083, rx=-0.000, ry=0.000, rz=-0.000, shoulder=lefty, elbow=epositive, wrist=wpositive, fatherId=fReference[0]}
  [528] = {x=-22.482, y=0.000, z=-4.093, rx=-0.000, ry=0.000, rz=-0.000, shoulder=lefty, elbow=epositive, wrist=wpositive, fatherId=fReference[0]}
  [529] = {x=-22.979, y=0.000, z=-4.102, rx=-0.000, ry=0.000, rz=-0.000, shoulder=lefty, elbow=epositive, wrist=wpositive, fatherId=fReference[0]}
  [530] = {x=-23.479, y=0.000, z=-4.111, rx=-0.000, ry=0.000, rz=-0.000, shoulder=lefty, elbow=epositive, wrist=wpositive, fatherId=fReference[0]}
  [531] = {x=-23.977, y=0.000, z=-4.121, rx=-0.000, ry=0.000, rz=-0.000, shoulder=lefty, elbow=epositive, wrist=wpositive, fatherId=fReference[0]}
  [532] = {x=-24.472, y=0.000, z=-4.131, rx=-0.000, ry=0.000, rz=-0.000, shoulder=lefty, elbow=epositive, wrist=wpositive, fatherId=fReference[0]}
  [533] = {x=-24.970, y=0.000, z=-4.141, rx=-0.000, ry=0.000, rz=-0.000, shoulder=lefty, elbow=epositive, wrist=wpositive, fatherId=fReference[0]}
  [534] = {x=-25.465, y=0.000, z=-4.151, rx=-0.000, ry=0.000, rz=-0.000, shoulder=lefty, elbow=epositive, wrist=wpositive, fatherId=fReference[0]}
  [535] = {x=-25.962, y=0.000, z=-4.161, rx=-0.000, ry=0.000, rz=-0.000, shoulder=lefty, elbow=epositive, wrist=wpositive, fatherId=fReference[0]}
  [536] = {x=-26.457, y=0.000, z=-4.171, rx=-0.000, ry=0.000, rz=-0.000, shoulder=lefty, elbow=epositive, wrist=wpositive, fatherId=fReference[0]}
  [537] = {x=-26.952, y=0.000, z=-4.181, rx=-0.000, ry=0.000, rz=-0.000, shoulder=lefty, elbow=epositive, wrist=wpositive, fatherId=fReference[0]}
  [538] = {x=-27.448, y=0.000, z=-4.191, rx=-0.000, ry=0.000, rz=-0.000, shoulder=lefty, elbow=epositive, wrist=wpositive, fatherId=fReference[0]}
  [539] = {x=-27.944, y=0.000, z=-4.201, rx=-0.000, ry=0.000, rz=-0.000, shoulder=lefty, elbow=epositive, wrist=wpositive, fatherId=fReference[0]}
  [540] = {x=-28.440, y=0.000, z=-4.212, rx=-0.000, ry=0.000, rz=-0.000, shoulder=lefty, elbow=epositive, wrist=wpositive, fatherId=fReference[0]}
  [541] = {x=-28.936, y=0.000, z=-4.222, rx=-0.000, ry=0.000, rz=-0.000, shoulder=lefty, elbow=epositive, wrist=wpositive, fatherId=fReference[0]}
  [542] = {x=-29.432, y=0.000, z=-4.232, rx=-0.000, ry=0.000, rz=-0.000, shoulder=lefty, elbow=epositive, wrist=wpositive, fatherId=fReference[0]}
  [543] = {x=-29.928, y=0.000, z=-4.242, rx=-0.000, ry=0.000, rz=-0.000, shoulder=lefty, elbow=epositive, wrist=wpositive, fatherId=fReference[0]}
  [544] = {x=-30.425, y=0.000, z=-4.252, rx=-0.000, ry=0.000, rz=-0.000, shoulder=lefty, elbow=epositive, wrist=wpositive, fatherId=fReference[0]}
  [545] = {x=-30.922, y=0.000, z=-4.262, rx=-0.000, ry=0.000, rz=-0.000, shoulder=lefty, elbow=epositive, wrist=wpositive, fatherId=fReference[0]}
  [546] = {x=-31.422, y=0.000, z=-4.272, rx=-0.000, ry=0.000, rz=-0.000, shoulder=lefty, elbow=epositive, wrist=wpositive, fatherId=fReference[0]}
  [547] = {x=-31.923, y=0.000, z=-4.282, rx=-0.000, ry=0.000, rz=-0.000, shoulder=lefty, elbow=epositive, wrist=wpositive, fatherId=fReference[0]}
  [548] = {x=-32.429, y=0.000, z=-4.291, rx=-0.000, ry=0.000, rz=-0.000, shoulder=lefty, elbow=epositive, wrist=wpositive, fatherId=fReference[0]}
  [549] = {x=-31.749, y=0.000, z=-4.264, rx=-0.000, ry=0.000, rz=-0.000, shoulder=lefty, elbow=epositive, wrist=wpositive, fatherId=fReference[0]}
  [550] = {x=-31.249, y=0.000, z=-4.258, rx=-0.000, ry=0.000, rz=-0.000, shoulder=lefty, elbow=epositive, wrist=wpositive, fatherId=fReference[0]}
  [551] = {x=-30.754, y=0.000, z=-4.258, rx=-0.000, ry=0.000, rz=-0.000, shoulder=lefty, elbow=epositive, wrist=wpositive, fatherId=fReference[0]}
  [552] = {x=-30.259, y=0.000, z=-4.259, rx=-0.000, ry=0.000, rz=-0.000, shoulder=lefty, elbow=epositive, wrist=wpositive, fatherId=fReference[0]}
  [553] = {x=-29.762, y=0.000, z=-4.263, rx=-0.000, ry=0.000, rz=-0.000, shoulder=lefty, elbow=epositive, wrist=wpositive, fatherId=fReference[0]}
  [554] = {x=-29.262, y=0.000, z=-4.268, rx=-0.000, ry=0.000, rz=-0.000, shoulder=lefty, elbow=epositive, wrist=wpositive, fatherId=fReference[0]}
  [555] = {x=-28.763, y=0.000, z=-4.274, rx=-0.000, ry=0.000, rz=-0.000, shoulder=lefty, elbow=epositive, wrist=wpositive, fatherId=fReference[0]}
  [556] = {x=-28.262, y=0.000, z=-4.281, rx=-0.000, ry=0.000, rz=-0.000, shoulder=lefty, elbow=epositive, wrist=wpositive, fatherId=fReference[0]}
  [557] = {x=-27.760, y=0.000, z=-4.288, rx=-0.000, ry=0.000, rz=-0.000, shoulder=lefty, elbow=epositive, wrist=wpositive, fatherId=fReference[0]}
  [558] = {x=-27.260, y=0.000, z=-4.295, rx=-0.000, ry=0.000, rz=-0.000, shoulder=lefty, elbow=epositive, wrist=wpositive, fatherId=fReference[0]}
  [559] = {x=-26.758, y=0.000, z=-4.303, rx=-0.000, ry=0.000, rz=-0.000, shoulder=lefty, elbow=epositive, wrist=wpositive, fatherId=fReference[0]}
  [560] = {x=-26.256, y=0.000, z=-4.310, rx=-0.000, ry=0.000, rz=-0.000, shoulder=lefty, elbow=epositive, wrist=wpositive, fatherId=fReference[0]}
  [561] = {x=-25.754, y=0.000, z=-4.318, rx=-0.000, ry=0.000, rz=-0.000, shoulder=lefty, elbow=epositive, wrist=wpositive, fatherId=fReference[0]}
  [562] = {x=-25.252, y=0.000, z=-4.326, rx=-0.000, ry=0.000, rz=-0.000, shoulder=lefty, elbow=epositive, wrist=wpositive, fatherId=fReference[0]}
  [563] = {x=-24.748, y=0.000, z=-4.334, rx=-0.000, ry=0.000, rz=-0.000, shoulder=lefty, elbow=epositive, wrist=wpositive, fatherId=fReference[0]}
  [564] = {x=-24.246, y=0.000, z=-4.342, rx=-0.000, ry=0.000, rz=-0.000, shoulder=lefty, elbow=epositive, wrist=wpositive, fatherId=fReference[0]}
  [565] = {x=-23.741, y=0.000, z=-4.350, rx=-0.000, ry=0.000, rz=-0.000, shoulder=lefty, elbow=epositive, wrist=wpositive, fatherId=fReference[0]}
  [566] = {x=-23.238, y=0.000, z=-4.359, rx=-0.000, ry=0.000, rz=-0.000, shoulder=lefty, elbow=epositive, wrist=wpositive, fatherId=fReference[0]}
  [567] = {x=-22.734, y=0.000, z=-4.367, rx=-0.000, ry=0.000, rz=-0.000, shoulder=lefty, elbow=epositive, wrist=wpositive, fatherId=fReference[0]}
  [568] = {x=-22.230, y=0.000, z=-4.376, rx=-0.000, ry=0.000, rz=-0.000, shoulder=lefty, elbow=epositive, wrist=wpositive, fatherId=fReference[0]}
  [569] = {x=-21.725, y=0.000, z=-4.384, rx=-0.000, ry=0.000, rz=-0.000, shoulder=lefty, elbow=epositive, wrist=wpositive, fatherId=fReference[0]}
  [570] = {x=-21.221, y=0.000, z=-4.393, rx=-0.000, ry=0.000, rz=-0.000, shoulder=lefty, elbow=epositive, wrist=wpositive, fatherId=fReference[0]}
  [571] = {x=-20.717, y=0.000, z=-4.402, rx=-0.000, ry=0.000, rz=-0.000, shoulder=lefty, elbow=epositive, wrist=wpositive, fatherId=fReference[0]}
  [572] = {x=-20.213, y=0.000, z=-4.410, rx=-0.000, ry=0.000, rz=-0.000, shoulder=lefty, elbow=epositive, wrist=wpositive, fatherId=fReference[0]}
  [573] = {x=-19.709, y=0.000, z=-4.419, rx=-0.000, ry=0.000, rz=-0.000, shoulder=lefty, elbow=epositive, wrist=wpositive, fatherId=fReference[0]}
  [574] = {x=-19.205, y=0.000, z=-4.427, rx=-0.000, ry=0.000, rz=-0.000, shoulder=lefty, elbow=epositive, wrist=wpositive, fatherId=fReference[0]}
  [575] = {x=-18.701, y=0.000, z=-4.436, rx=-0.000, ry=0.000, rz=-0.000, shoulder=lefty, elbow=epositive, wrist=wpositive, fatherId=fReference[0]}
  [576] = {x=-18.197, y=0.000, z=-4.444, rx=-0.000, ry=0.000, rz=-0.000, shoulder=lefty, elbow=epositive, wrist=wpositive, fatherId=fReference[0]}
  [577] = {x=-17.692, y=0.000, z=-4.452, rx=-0.000, ry=0.000, rz=-0.000, shoulder=lefty, elbow=epositive, wrist=wpositive, fatherId=fReference[0]}
  [578] = {x=-17.189, y=0.000, z=-4.461, rx=-0.000, ry=0.000, rz=-0.000, shoulder=lefty, elbow=epositive, wrist=wpositive, fatherId=fReference[0]}
  [579] = {x=-16.685, y=0.000, z=-4.469, rx=-0.000, ry=0.000, rz=-0.000, shoulder=lefty, elbow=epositive, wrist=wpositive, fatherId=fReference[0]}
  [580] = {x=-16.180, y=0.000, z=-4.477, rx=-0.000, ry=0.000, rz=-0.000, shoulder=lefty, elbow=epositive, wrist=wpositive, fatherId=fReference[0]}
  [581] = {x=-15.676, y=0.000, z=-4.486, rx=-0.000, ry=0.000, rz=-0.000, shoulder=lefty, elbow=epositive, wrist=wpositive, fatherId=fReference[0]}
  [582] = {x=-15.172, y=0.000, z=-4.494, rx=-0.000, ry=0.000, rz=-0.000, shoulder=lefty, elbow=epositive, wrist=wpositive, fatherId=fReference[0]}
  [583] = {x=-14.669, y=0.000, z=-4.502, rx=-0.000, ry=0.000, rz=-0.000, shoulder=lefty, elbow=epositive, wrist=wpositive, fatherId=fReference[0]}
  [584] = {x=-14.166, y=0.000, z=-4.511, rx=-0.000, ry=0.000, rz=-0.000, shoulder=lefty, elbow=epositive, wrist=wpositive, fatherId=fReference[0]}
  [585] = {x=-13.663, y=0.000, z=-4.519, rx=-0.000, ry=0.000, rz=-0.000, shoulder=lefty, elbow=epositive, wrist=wpositive, fatherId=fReference[0]}
  [586] = {x=-13.160, y=0.000, z=-4.526, rx=-0.000, ry=0.000, rz=-0.000, shoulder=lefty, elbow=epositive, wrist=wpositive, fatherId=fReference[0]}
  [587] = {x=-12.657, y=0.000, z=-4.534, rx=-0.000, ry=0.000, rz=-0.000, shoulder=lefty, elbow=epositive, wrist=wpositive, fatherId=fReference[0]}
  [588] = {x=-12.154, y=0.000, z=-4.542, rx=-0.000, ry=0.000, rz=-0.000, shoulder=lefty, elbow=epositive, wrist=wpositive, fatherId=fReference[0]}
  [589] = {x=-11.652, y=0.000, z=-4.550, rx=-0.000, ry=0.000, rz=-0.000, shoulder=lefty, elbow=epositive, wrist=wpositive, fatherId=fReference[0]}
  [590] = {x=-11.149, y=0.000, z=-4.558, rx=-0.000, ry=0.000, rz=-0.000, shoulder=lefty, elbow=epositive, wrist=wpositive, fatherId=fReference[0]}
  [591] = {x=-10.646, y=0.000, z=-4.566, rx=-0.000, ry=0.000, rz=-0.000, shoulder=lefty, elbow=epositive, wrist=wpositive, fatherId=fReference[0]}
  [592] = {x=-10.143, y=0.000, z=-4.574, rx=-0.000, ry=0.000, rz=-0.000, shoulder=lefty, elbow=epositive, wrist=wpositive, fatherId=fReference[0]}
  [593] = {x=-9.640, y=0.000, z=-4.582, rx=-0.000, ry=0.000, rz=-0.000, shoulder=lefty, elbow=epositive, wrist=wpositive, fatherId=fReference[0]}
  [594] = {x=-9.137, y=0.000, z=-4.590, rx=-0.000, ry=0.000, rz=-0.000, shoulder=lefty, elbow=epositive, wrist=wpositive, fatherId=fReference[0]}
  [595] = {x=-8.634, y=0.000, z=-4.598, rx=-0.000, ry=0.000, rz=-0.000, shoulder=lefty, elbow=epositive, wrist=wpositive, fatherId=fReference[0]}
  [596] = {x=-8.132, y=0.000, z=-4.605, rx=-0.000, ry=0.000, rz=-0.000, shoulder=lefty, elbow=epositive, wrist=wpositive, fatherId=fReference[0]}
  [597] = {x=-7.630, y=0.000, z=-4.613, rx=-0.000, ry=0.000, rz=-0.000, shoulder=lefty, elbow=epositive, wrist=wpositive, fatherId=fReference[0]}
  [598] = {x=-7.128, y=0.000, z=-4.621, rx=-0.000, ry=0.000, rz=-0.000, shoulder=lefty, elbow=epositive, wrist=wpositive, fatherId=fReference[0]}
  [599] = {x=-6.625, y=0.000, z=-4.629, rx=-0.000, ry=0.000, rz=-0.000, shoulder=lefty, elbow=epositive, wrist=wpositive, fatherId=fReference[0]}
  [600] = {x=-6.123, y=0.000, z=-4.636, rx=-0.000, ry=0.000, rz=-0.000, shoulder=lefty, elbow=epositive, wrist=wpositive, fatherId=fReference[0]}
  [601] = {x=-5.621, y=0.000, z=-4.644, rx=-0.000, ry=0.000, rz=-0.000, shoulder=lefty, elbow=epositive, wrist=wpositive, fatherId=fReference[0]}
  [602] = {x=-5.118, y=0.000, z=-4.652, rx=-0.000, ry=0.000, rz=-0.000, shoulder=lefty, elbow=epositive, wrist=wpositive, fatherId=fReference[0]}
  [603] = {x=-4.616, y=0.000, z=-4.660, rx=-0.000, ry=0.000, rz=-0.000, shoulder=lefty, elbow=epositive, wrist=wpositive, fatherId=fReference[0]}
  [604] = {x=-4.114, y=0.000, z=-4.667, rx=-0.000, ry=0.000, rz=-0.000, shoulder=lefty, elbow=epositive, wrist=wpositive, fatherId=fReference[0]}
  [605] = {x=-3.612, y=0.000, z=-4.675, rx=-0.000, ry=0.000, rz=-0.000, shoulder=lefty, elbow=epositive, wrist=wpositive, fatherId=fReference[0]}
  [606] = {x=-3.110, y=0.000, z=-4.682, rx=-0.000, ry=0.000, rz=-0.000, shoulder=lefty, elbow=epositive, wrist=wpositive, fatherId=fReference[0]}
  [607] = {x=-2.608, y=0.000, z=-4.690, rx=-0.000, ry=0.000, rz=-0.000, shoulder=lefty, elbow=epositive, wrist=wpositive, fatherId=fReference[0]}
  [608] = {x=-2.105, y=0.000, z=-4.698, rx=-0.000, ry=0.000, rz=-0.000, shoulder=lefty, elbow=epositive, wrist=wpositive, fatherId=fReference[0]}
  [609] = {x=-1.603, y=0.000, z=-4.705, rx=-0.000, ry=0.000, rz=-0.000, shoulder=lefty, elbow=epositive, wrist=wpositive, fatherId=fReference[0]}
  [610] = {x=-1.100, y=0.000, z=-4.713, rx=-0.000, ry=0.000, rz=-0.000, shoulder=lefty, elbow=epositive, wrist=wpositive, fatherId=fReference[0]}
  [611] = {x=-0.598, y=0.000, z=-4.721, rx=-0.000, ry=0.000, rz=-0.000, shoulder=lefty, elbow=epositive, wrist=wpositive, fatherId=fReference[0]}
  [612] = {x=-0.095, y=0.000, z=-4.729, rx=-0.000, ry=0.000, rz=-0.000, shoulder=lefty, elbow=epositive, wrist=wpositive, fatherId=fReference[0]}
  [613] = {x=0.409, y=0.000, z=-4.737, rx=-0.000, ry=0.000, rz=-0.000, shoulder=lefty, elbow=epositive, wrist=wpositive, fatherId=fReference[0]}
  [614] = {x=0.912, y=0.000, z=-4.745, rx=-0.000, ry=0.000, rz=-0.000, shoulder=lefty, elbow=epositive, wrist=wpositive, fatherId=fReference[0]}
  [615] = {x=1.416, y=0.000, z=-4.753, rx=-0.000, ry=0.000, rz=-0.000, shoulder=lefty, elbow=epositive, wrist=wpositive, fatherId=fReference[0]}
  [616] = {x=1.920, y=0.000, z=-4.761, rx=-0.000, ry=0.000, rz=-0.000, shoulder=lefty, elbow=epositive, wrist=wpositive, fatherId=fReference[0]}
  [617] = {x=2.423, y=0.000, z=-4.770, rx=-0.000, ry=0.000, rz=-0.000, shoulder=lefty, elbow=epositive, wrist=wpositive, fatherId=fReference[0]}
  [618] = {x=2.927, y=0.000, z=-4.777, rx=-0.000, ry=0.000, rz=-0.000, shoulder=lefty, elbow=epositive, wrist=wpositive, fatherId=fReference[0]}
  [619] = {x=3.430, y=0.000, z=-4.785, rx=-0.000, ry=0.000, rz=-0.000, shoulder=lefty, elbow=epositive, wrist=wpositive, fatherId=fReference[0]}
  [620] = {x=3.934, y=0.000, z=-4.792, rx=-0.000, ry=0.000, rz=-0.000, shoulder=lefty, elbow=epositive, wrist=wpositive, fatherId=fReference[0]}
  [621] = {x=4.438, y=0.000, z=-4.800, rx=-0.000, ry=0.000, rz=-0.000, shoulder=lefty, elbow=epositive, wrist=wpositive, fatherId=fReference[0]}
  [622] = {x=4.942, y=0.000, z=-4.808, rx=-0.000, ry=0.000, rz=-0.000, shoulder=lefty, elbow=epositive, wrist=wpositive, fatherId=fReference[0]}
  [623] = {x=5.447, y=0.000, z=-4.816, rx=-0.000, ry=0.000, rz=-0.000, shoulder=lefty, elbow=epositive, wrist=wpositive, fatherId=fReference[0]}
  [624] = {x=5.951, y=0.000, z=-4.825, rx=-0.000, ry=0.000, rz=-0.000, shoulder=lefty, elbow=epositive, wrist=wpositive, fatherId=fReference[0]}
  [625] = {x=6.456, y=0.000, z=-4.833, rx=-0.000, ry=0.000, rz=-0.000, shoulder=lefty, elbow=epositive, wrist=wpositive, fatherId=fReference[0]}
  [626] = {x=6.960, y=0.000, z=-4.841, rx=-0.000, ry=0.000, rz=-0.000, shoulder=lefty, elbow=epositive, wrist=wpositive, fatherId=fReference[0]}
  [627] = {x=7.464, y=0.000, z=-4.849, rx=-0.000, ry=0.000, rz=-0.000, shoulder=lefty, elbow=epositive, wrist=wpositive, fatherId=fReference[0]}
  [628] = {x=7.969, y=0.000, z=-4.857, rx=-0.000, ry=0.000, rz=-0.000, shoulder=lefty, elbow=epositive, wrist=wpositive, fatherId=fReference[0]}
  [629] = {x=8.474, y=0.000, z=-4.866, rx=-0.000, ry=0.000, rz=-0.000, shoulder=lefty, elbow=epositive, wrist=wpositive, fatherId=fReference[0]}
  [630] = {x=8.980, y=0.000, z=-4.874, rx=-0.000, ry=0.000, rz=-0.000, shoulder=lefty, elbow=epositive, wrist=wpositive, fatherId=fReference[0]}
  [631] = {x=9.485, y=0.000, z=-4.883, rx=-0.000, ry=0.000, rz=-0.000, shoulder=lefty, elbow=epositive, wrist=wpositive, fatherId=fReference[0]}
  [632] = {x=9.990, y=0.000, z=-4.891, rx=-0.000, ry=0.000, rz=-0.000, shoulder=lefty, elbow=epositive, wrist=wpositive, fatherId=fReference[0]}
  [633] = {x=10.496, y=0.000, z=-4.899, rx=-0.000, ry=0.000, rz=-0.000, shoulder=lefty, elbow=epositive, wrist=wpositive, fatherId=fReference[0]}
  [634] = {x=11.001, y=0.000, z=-4.908, rx=-0.000, ry=0.000, rz=-0.000, shoulder=lefty, elbow=epositive, wrist=wpositive, fatherId=fReference[0]}
  [635] = {x=11.508, y=0.000, z=-4.917, rx=-0.000, ry=0.000, rz=-0.000, shoulder=lefty, elbow=epositive, wrist=wpositive, fatherId=fReference[0]}
  [636] = {x=12.014, y=0.000, z=-4.925, rx=-0.000, ry=0.000, rz=-0.000, shoulder=lefty, elbow=epositive, wrist=wpositive, fatherId=fReference[0]}
  [637] = {x=12.520, y=0.000, z=-4.934, rx=-0.000, ry=0.000, rz=-0.000, shoulder=lefty, elbow=epositive, wrist=wpositive, fatherId=fReference[0]}
  [638] = {x=13.027, y=0.000, z=-4.943, rx=-0.000, ry=0.000, rz=-0.000, shoulder=lefty, elbow=epositive, wrist=wpositive, fatherId=fReference[0]}
  [639] = {x=13.534, y=0.000, z=-4.951, rx=-0.000, ry=0.000, rz=-0.000, shoulder=lefty, elbow=epositive, wrist=wpositive, fatherId=fReference[0]}
  [640] = {x=14.040, y=0.000, z=-4.960, rx=-0.000, ry=0.000, rz=-0.000, shoulder=lefty, elbow=epositive, wrist=wpositive, fatherId=fReference[0]}
  [641] = {x=14.547, y=0.000, z=-4.969, rx=-0.000, ry=0.000, rz=-0.000, shoulder=lefty, elbow=epositive, wrist=wpositive, fatherId=fReference[0]}
  [642] = {x=15.054, y=0.000, z=-4.978, rx=-0.000, ry=0.000, rz=-0.000, shoulder=lefty, elbow=epositive, wrist=wpositive, fatherId=fReference[0]}
  [643] = {x=15.562, y=0.000, z=-4.987, rx=-0.000, ry=0.000, rz=-0.000, shoulder=lefty, elbow=epositive, wrist=wpositive, fatherId=fReference[0]}
  [644] = {x=16.069, y=0.000, z=-4.996, rx=-0.000, ry=0.000, rz=-0.000, shoulder=lefty, elbow=epositive, wrist=wpositive, fatherId=fReference[0]}
  [645] = {x=16.576, y=0.000, z=-5.005, rx=-0.000, ry=0.000, rz=-0.000, shoulder=lefty, elbow=epositive, wrist=wpositive, fatherId=fReference[0]}
  [646] = {x=17.083, y=0.000, z=-5.013, rx=-0.000, ry=0.000, rz=-0.000, shoulder=lefty, elbow=epositive, wrist=wpositive, fatherId=fReference[0]}
  [647] = {x=17.590, y=0.000, z=-5.022, rx=-0.000, ry=0.000, rz=-0.000, shoulder=lefty, elbow=epositive, wrist=wpositive, fatherId=fReference[0]}
  [648] = {x=18.100, y=0.000, z=-5.032, rx=-0.000, ry=0.000, rz=-0.000, shoulder=lefty, elbow=epositive, wrist=wpositive, fatherId=fReference[0]}
  [649] = {x=18.607, y=0.000, z=-5.041, rx=-0.000, ry=0.000, rz=-0.000, shoulder=lefty, elbow=epositive, wrist=wpositive, fatherId=fReference[0]}
  [650] = {x=19.114, y=0.000, z=-5.050, rx=-0.000, ry=0.000, rz=-0.000, shoulder=lefty, elbow=epositive, wrist=wpositive, fatherId=fReference[0]}
  [651] = {x=19.622, y=0.000, z=-5.059, rx=-0.000, ry=0.000, rz=-0.000, shoulder=lefty, elbow=epositive, wrist=wpositive, fatherId=fReference[0]}
  [652] = {x=20.131, y=0.000, z=-5.069, rx=-0.000, ry=0.000, rz=-0.000, shoulder=lefty, elbow=epositive, wrist=wpositive, fatherId=fReference[0]}
  [653] = {x=20.640, y=0.000, z=-5.078, rx=-0.000, ry=0.000, rz=-0.000, shoulder=lefty, elbow=epositive, wrist=wpositive, fatherId=fReference[0]}
  [654] = {x=21.149, y=0.000, z=-5.088, rx=-0.000, ry=0.000, rz=-0.000, shoulder=lefty, elbow=epositive, wrist=wpositive, fatherId=fReference[0]}
  [655] = {x=21.659, y=0.000, z=-5.098, rx=-0.000, ry=0.000, rz=-0.000, shoulder=lefty, elbow=epositive, wrist=wpositive, fatherId=fReference[0]}
  [656] = {x=22.168, y=0.000, z=-5.107, rx=-0.000, ry=0.000, rz=-0.000, shoulder=lefty, elbow=epositive, wrist=wpositive, fatherId=fReference[0]}
  [657] = {x=22.677, y=0.000, z=-5.117, rx=-0.000, ry=0.000, rz=-0.000, shoulder=lefty, elbow=epositive, wrist=wpositive, fatherId=fReference[0]}
  [658] = {x=23.187, y=0.000, z=-5.127, rx=-0.000, ry=0.000, rz=-0.000, shoulder=lefty, elbow=epositive, wrist=wpositive, fatherId=fReference[0]}
  [659] = {x=23.697, y=0.000, z=-5.137, rx=-0.000, ry=0.000, rz=-0.000, shoulder=lefty, elbow=epositive, wrist=wpositive, fatherId=fReference[0]}
  [660] = {x=24.207, y=0.000, z=-5.147, rx=-0.000, ry=0.000, rz=-0.000, shoulder=lefty, elbow=epositive, wrist=wpositive, fatherId=fReference[0]}
  [661] = {x=24.717, y=0.000, z=-5.157, rx=-0.000, ry=0.000, rz=-0.000, shoulder=lefty, elbow=epositive, wrist=wpositive, fatherId=fReference[0]}
  [662] = {x=25.227, y=0.000, z=-5.167, rx=-0.000, ry=0.000, rz=-0.000, shoulder=lefty, elbow=epositive, wrist=wpositive, fatherId=fReference[0]}
  [663] = {x=25.738, y=0.000, z=-5.177, rx=-0.000, ry=0.000, rz=-0.000, shoulder=lefty, elbow=epositive, wrist=wpositive, fatherId=fReference[0]}
  [664] = {x=26.249, y=0.000, z=-5.187, rx=-0.000, ry=0.000, rz=-0.000, shoulder=lefty, elbow=epositive, wrist=wpositive, fatherId=fReference[0]}
  [665] = {x=26.761, y=0.000, z=-5.197, rx=-0.000, ry=0.000, rz=-0.000, shoulder=lefty, elbow=epositive, wrist=wpositive, fatherId=fReference[0]}
  [666] = {x=27.273, y=0.000, z=-5.207, rx=-0.000, ry=0.000, rz=-0.000, shoulder=lefty, elbow=epositive, wrist=wpositive, fatherId=fReference[0]}
  [667] = {x=27.785, y=0.000, z=-5.217, rx=-0.000, ry=0.000, rz=-0.000, shoulder=lefty, elbow=epositive, wrist=wpositive, fatherId=fReference[0]}
  [668] = {x=28.298, y=0.000, z=-5.227, rx=-0.000, ry=0.000, rz=-0.000, shoulder=lefty, elbow=epositive, wrist=wpositive, fatherId=fReference[0]}
  [669] = {x=28.811, y=0.000, z=-5.237, rx=-0.000, ry=0.000, rz=-0.000, shoulder=lefty, elbow=epositive, wrist=wpositive, fatherId=fReference[0]}
  [670] = {x=29.325, y=0.000, z=-5.248, rx=-0.000, ry=0.000, rz=-0.000, shoulder=lefty, elbow=epositive, wrist=wpositive, fatherId=fReference[0]}
  [671] = {x=29.838, y=0.000, z=-5.258, rx=-0.000, ry=0.000, rz=-0.000, shoulder=lefty, elbow=epositive, wrist=wpositive, fatherId=fReference[0]}
  [672] = {x=30.351, y=0.000, z=-5.268, rx=-0.000, ry=0.000, rz=-0.000, shoulder=lefty, elbow=epositive, wrist=wpositive, fatherId=fReference[0]}
  [673] = {x=30.865, y=0.000, z=-5.277, rx=-0.000, ry=0.000, rz=-0.000, shoulder=lefty, elbow=epositive, wrist=wpositive, fatherId=fReference[0]}
  [674] = {x=31.379, y=0.000, z=-5.287, rx=-0.000, ry=0.000, rz=-0.000, shoulder=lefty, elbow=epositive, wrist=wpositive, fatherId=fReference[0]}
  [675] = {x=31.897, y=0.000, z=-5.296, rx=-0.000, ry=0.000, rz=-0.000, shoulder=lefty, elbow=epositive, wrist=wpositive, fatherId=fReference[0]}
  [676] = {x=32.411, y=0.000, z=-5.305, rx=-0.000, ry=0.000, rz=-0.000, shoulder=lefty, elbow=epositive, wrist=wpositive, fatherId=fReference[0]}
  [677] = {x=32.924, y=0.000, z=-5.312, rx=-0.000, ry=0.000, rz=-0.000, shoulder=lefty, elbow=epositive, wrist=wpositive, fatherId=fReference[0]}
  [678] = {x=33.434, y=0.000, z=-5.318, rx=-0.000, ry=0.000, rz=-0.000, shoulder=lefty, elbow=epositive, wrist=wpositive, fatherId=fReference[0]}
  [679] = {x=33.948, y=0.000, z=-5.324, rx=-0.000, ry=0.000, rz=-0.000, shoulder=lefty, elbow=epositive, wrist=wpositive, fatherId=fReference[0]}
